       #MyWord := W#0;
       #MyBoolsinWord[8] := #"EMUOK";    //EPICSName: EMUOK
       #MyBoolsinWord[9] := #"EMUOK_Magtr";    //EPICSName: EMUOK_Magtr
       "PLCToEPICS"."Word"[#PLCToEPICSDataBlockOffset + 0] := #MyWord;
    Else
       #DEVICE_PARAM_OK := FALSE; //Invalid Hash
    END_IF;
END_FUNCTION_BLOCK
FUNCTION_BLOCK "DEVTYPE_ISRC_LEBT_INTF_HMI"
{ S7_Optimized_Access := 'TRUE' }
VERSION : 1.0
   VAR_INPUT
      "ComIocOK" { ExternalAccessible := 'True'; ExternalVisible := 'False'; ExternalWritable := 'False'; } : BOOL;   //EPICS Status variable: ComIocOK
      "ComRioOK" { ExternalAccessible := 'True'; ExternalVisible := 'False'; ExternalWritable := 'False'; } : BOOL;   //EPICS Status variable: ComRioOK
      "ISrcOK" { ExternalAccessible := 'True'; ExternalVisible := 'False'; ExternalWritable := 'False'; } : BOOL;   //EPICS Status variable: ISrcOK
      "EVENT_A_MEMO" { ExternalAccessible := 'True'; ExternalVisible := 'False'; ExternalWritable := 'False'; } : BOOL;   //EPICS Status variable: EVENT_A_MEMO
      "EVENT_B_MEMO" { ExternalAccessible := 'True'; ExternalVisible := 'False'; ExternalWritable := 'False'; } : BOOL;   //EPICS Status variable: EVENT_B_MEMO
      "EVENT_C_MEMO" { ExternalAccessible := 'True'; ExternalVisible := 'False'; ExternalWritable := 'False'; } : BOOL;   //EPICS Status variable: EVENT_C_MEMO
      "EVENT_D_MEMO" { ExternalAccessible := 'True'; ExternalVisible := 'False'; ExternalWritable := 'False'; } : BOOL;   //EPICS Status variable: EVENT_D_MEMO
      "EVENT_E_MEMO" { ExternalAccessible := 'True'; ExternalVisible := 'False'; ExternalWritable := 'False'; } : BOOL;   //EPICS Status variable: EVENT_E_MEMO
      "EVENT_F_MEMO" { ExternalAccessible := 'True'; ExternalVisible := 'False'; ExternalWritable := 'False'; } : BOOL;   //EPICS Status variable: EVENT_F_MEMO
      "EVENT_G_MEMO" { ExternalAccessible := 'True'; ExternalVisible := 'False'; ExternalWritable := 'False'; } : BOOL;   //EPICS Status variable: EVENT_G_MEMO
      "EVENT_H_MEMO" { ExternalAccessible := 'True'; ExternalVisible := 'False'; ExternalWritable := 'False'; } : BOOL;   //EPICS Status variable: EVENT_H_MEMO
      "ChopPwrSysOK_MEMO" { ExternalAccessible := 'True'; ExternalVisible := 'False'; ExternalWritable := 'False'; } : BOOL;   //EPICS Status variable: ChopPwrSysOK_MEMO
      "ChopVoltAlarm_MEMO" { ExternalAccessible := 'True'; ExternalVisible := 'False'; ExternalWritable := 'False'; } : BOOL;   //EPICS Status variable: ChopVoltAlarm_MEMO
      "ChopWtrFlowOK_MEMO" { ExternalAccessible := 'True'; ExternalVisible := 'False'; ExternalWritable := 'False'; } : BOOL;   //EPICS Status variable: ChopWtrFlowOK_MEMO
      "Sol1WtrTempOK_MEMO" { ExternalAccessible := 'True'; ExternalVisible := 'False'; ExternalWritable := 'False'; } : BOOL;   //EPICS Status variable: Sol1WtrTempOK_MEMO
      "Sol2WtrTempOK_MEMO" { ExternalAccessible := 'True'; ExternalVisible := 'False'; ExternalWritable := 'False'; } : BOOL;   //EPICS Status variable: Sol2WtrTempOK_MEMO
      "Sol1WtrFlowOK_MEMO" { ExternalAccessible := 'True'; ExternalVisible := 'False'; ExternalWritable := 'False'; } : BOOL;   //EPICS Status variable: Sol1WtrFlowOK_MEMO
      "Sol2WtrFlowOK_MEMO" { ExternalAccessible := 'True'; ExternalVisible := 'False'; ExternalWritable := 'False'; } : BOOL;   //EPICS Status variable: Sol2WtrFlowOK_MEMO
      "Sol1CurMaxErr_MEMO" { ExternalAccessible := 'True'; ExternalVisible := 'False'; ExternalWritable := 'False'; } : BOOL;   //EPICS Status variable: Sol1CurMaxErr_MEMO
      "Sol2CurMaxErr_MEMO" { ExternalAccessible := 'True'; ExternalVisible := 'False'; ExternalWritable := 'False'; } : BOOL;   //EPICS Status variable: Sol2CurMaxErr_MEMO
      "Str1HCurMaxErr_MEMO" { ExternalAccessible := 'True'; ExternalVisible := 'False'; ExternalWritable := 'False'; } : BOOL;   //EPICS Status variable: Str1HCurMaxErr_MEMO
      "Str2HCurMaxErr_MEMO" { ExternalAccessible := 'True'; ExternalVisible := 'False'; ExternalWritable := 'False'; } : BOOL;   //EPICS Status variable: Str2HCurMaxErr_MEMO
      "Str1VCurMaxErr_MEMO" { ExternalAccessible := 'True'; ExternalVisible := 'False'; ExternalWritable := 'False'; } : BOOL;   //EPICS Status variable: Str1VCurMaxErr_MEMO
      "Str2VCurMaxErr_MEMO" { ExternalAccessible := 'True'; ExternalVisible := 'False'; ExternalWritable := 'False'; } : BOOL;   //EPICS Status variable: Str2VCurMaxErr_MEMO
      "Coil1PwrSuppOK_MEMO" { ExternalAccessible := 'True'; ExternalVisible := 'False'; ExternalWritable := 'False'; } : BOOL;   //EPICS Status variable: Coil1PwrSuppOK_MEMO
      "Coil2PwrSuppOK_MEMO" { ExternalAccessible := 'True'; ExternalVisible := 'False'; ExternalWritable := 'False'; } : BOOL;   //EPICS Status variable: Coil2PwrSuppOK_MEMO
      "Coil3PwrSuppOK_MEMO" { ExternalAccessible := 'True'; ExternalVisible := 'False'; ExternalWritable := 'False'; } : BOOL;   //EPICS Status variable: Coil3PwrSuppOK_MEMO
      "HVITLidOpenR_MEMO" { ExternalAccessible := 'True'; ExternalVisible := 'False'; ExternalWritable := 'False'; } : BOOL;   //EPICS Status variable: HVITLidOpenR_MEMO
      "HVITOilTempOK_MEMO" { ExternalAccessible := 'True'; ExternalVisible := 'False'; ExternalWritable := 'False'; } : BOOL;   //EPICS Status variable: HVITOilTempOK_MEMO
      "GndWtrTempMaxErr_MEMO" { ExternalAccessible := 'True'; ExternalVisible := 'False'; ExternalWritable := 'False'; } : BOOL;   //EPICS Status variable: GndWtrTempMaxErr_MEMO
      "HVWtrTempMaxErr_MEMO" { ExternalAccessible := 'True'; ExternalVisible := 'False'; ExternalWritable := 'False'; } : BOOL;   //EPICS Status variable: HVWtrTempMaxErr_MEMO
      "RepWtrFlowOK_MEMO" { ExternalAccessible := 'True'; ExternalVisible := 'False'; ExternalWritable := 'False'; } : BOOL;   //EPICS Status variable: RepWtrFlowOK_MEMO
      "IrisWtrTemp1Err_MEMO" { ExternalAccessible := 'True'; ExternalVisible := 'False'; ExternalWritable := 'False'; } : BOOL;   //EPICS Status variable: IrisWtrTemp1Err_MEMO
      "IrisWtrTemp2Err_MEMO" { ExternalAccessible := 'True'; ExternalVisible := 'False'; ExternalWritable := 'False'; } : BOOL;   //EPICS Status variable: IrisWtrTemp2Err_MEMO
      "IrisWtrFlowOK_MEMO" { ExternalAccessible := 'True'; ExternalVisible := 'False'; ExternalWritable := 'False'; } : BOOL;   //EPICS Status variable: IrisWtrFlowOK_MEMO
      "EMUHWtrFlowOK_MEMO" { ExternalAccessible := 'True'; ExternalVisible := 'False'; ExternalWritable := 'False'; } : BOOL;   //EPICS Status variable: EMUHWtrFlowOK_MEMO
      "EMUVWtrFlowOK_MEMO" { ExternalAccessible := 'True'; ExternalVisible := 'False'; ExternalWritable := 'False'; } : BOOL;   //EPICS Status variable: EMUVWtrFlowOK_MEMO
      "FCWtrFlowOK_MEMO" { ExternalAccessible := 'True'; ExternalVisible := 'False'; ExternalWritable := 'False'; } : BOOL;   //EPICS Status variable: FCWtrFlowOK_MEMO
      "EMUOK_MEMO" { ExternalAccessible := 'True'; ExternalVisible := 'False'; ExternalWritable := 'False'; } : BOOL;   //EPICS Status variable: EMUOK_MEMO
      "IBSWtrFlowOK_MEMO" { ExternalAccessible := 'True'; ExternalVisible := 'False'; ExternalWritable := 'False'; } : BOOL;   //EPICS Status variable: IBSWtrFlowOK_MEMO
      "CollWtrFlowOK_MEMO" { ExternalAccessible := 'True'; ExternalVisible := 'False'; ExternalWritable := 'False'; } : BOOL;   //EPICS Status variable: CollWtrFlowOK_MEMO
      "MatTrWtrFlowOK_MEMO" { ExternalAccessible := 'True'; ExternalVisible := 'False'; ExternalWritable := 'False'; } : BOOL;   //EPICS Status variable: MatTrWtrFlowOK_MEMO
      "PlasChWtrFlowOK_MEMO" { ExternalAccessible := 'True'; ExternalVisible := 'False'; ExternalWritable := 'False'; } : BOOL;   //EPICS Status variable: PlasChWtrFlowOK_MEMO
      "VacOK_MEMO" { ExternalAccessible := 'True'; ExternalVisible := 'False'; ExternalWritable := 'False'; } : BOOL;   //EPICS Status variable: VacOK_MEMO
      "VacPermit_MEMO" { ExternalAccessible := 'True'; ExternalVisible := 'False'; ExternalWritable := 'False'; } : BOOL;   //EPICS Status variable: VacPermit_MEMO
      "ComRioOK_MEMO" { ExternalAccessible := 'True'; ExternalVisible := 'False'; ExternalWritable := 'False'; } : BOOL;   //EPICS Status variable: ComRioOK_MEMO
      "MPSOK_MEMO" { ExternalAccessible := 'True'; ExternalVisible := 'False'; ExternalWritable := 'False'; } : BOOL;   //EPICS Status variable: MPSOK_MEMO
      "HVPSVolOK_Magtr_MEMO" { ExternalAccessible := 'True'; ExternalVisible := 'False'; ExternalWritable := 'False'; } : BOOL;   //EPICS Status variable: HVPSVolOK_Magtr_MEMO
      "DPLOK_MEMO" { ExternalAccessible := 'True'; ExternalVisible := 'False'; ExternalWritable := 'False'; } : BOOL;   //EPICS Status variable: DPLOK_MEMO
      "HVPfDoors_MEMO" { ExternalAccessible := 'True'; ExternalVisible := 'False'; ExternalWritable := 'False'; } : BOOL;   //EPICS Status variable: HVPfDoors_MEMO
      "HVPfRes_MEMO" { ExternalAccessible := 'True'; ExternalVisible := 'False'; ExternalWritable := 'False'; } : BOOL;   //EPICS Status variable: HVPfRes_MEMO
      "HVPermit_MEMO" { ExternalAccessible := 'True'; ExternalVisible := 'False'; ExternalWritable := 'False'; } : BOOL;   //EPICS Status variable: HVPermit_MEMO
      "ComIocOK_MEMO" { ExternalAccessible := 'True'; ExternalVisible := 'False'; ExternalWritable := 'False'; } : BOOL;   //EPICS Status variable: ComIocOK_MEMO
      "Rep1VolOK_MEMO" { ExternalAccessible := 'True'; ExternalVisible := 'False'; ExternalWritable := 'False'; } : BOOL;   //EPICS Status variable: Rep1VolOK_MEMO
      "Rep2VolOK_MEMO" { ExternalAccessible := 'True'; ExternalVisible := 'False'; ExternalWritable := 'False'; } : BOOL;   //EPICS Status variable: Rep2VolOK_MEMO
      "MagPulseModeOK_MEMO" { ExternalAccessible := 'True'; ExternalVisible := 'False'; ExternalWritable := 'False'; } : BOOL;   //EPICS Status variable: MagPulseModeOK_MEMO
      "ESTOP_MEMO" { ExternalAccessible := 'True'; ExternalVisible := 'False'; ExternalWritable := 'False'; } : BOOL;   //EPICS Status variable: ESTOP_MEMO
      "HVPSConnErr_MEMO" { ExternalAccessible := 'True'; ExternalVisible := 'False'; ExternalWritable := 'False'; } : BOOL;   //EPICS Status variable: HVPSConnErr_MEMO
      "Coil1WtrFlowOK_MEMO" { ExternalAccessible := 'True'; ExternalVisible := 'False'; ExternalWritable := 'False'; } : BOOL;   //EPICS Status variable: Coil1WtrFlowOK_MEMO
      "Coil2WtrFlowOK_MEMO" { ExternalAccessible := 'True'; ExternalVisible := 'False'; ExternalWritable := 'False'; } : BOOL;   //EPICS Status variable: Coil2WtrFlowOK_MEMO
      "Coil3WtrFlowOK_MEMO" { ExternalAccessible := 'True'; ExternalVisible := 'False'; ExternalWritable := 'False'; } : BOOL;   //EPICS Status variable: Coil3WtrFlowOK_MEMO
      "Coil1WtrTempOK_MEMO" { ExternalAccessible := 'True'; ExternalVisible := 'False'; ExternalWritable := 'False'; } : BOOL;   //EPICS Status variable: Coil1WtrTempOK_MEMO
      "Coil2WtrTempOK_MEMO" { ExternalAccessible := 'True'; ExternalVisible := 'False'; ExternalWritable := 'False'; } : BOOL;   //EPICS Status variable: Coil2WtrTempOK_MEMO
      "Coil3WtrTempOK_MEMO" { ExternalAccessible := 'True'; ExternalVisible := 'False'; ExternalWritable := 'False'; } : BOOL;   //EPICS Status variable: Coil3WtrTempOK_MEMO
      "F_MagtrEnCmd" { ExternalAccessible := 'True'; ExternalVisible := 'False'; ExternalWritable := 'False'; } : BOOL;   //EPICS Status variable: F_MagtrEnCmd
      "F_ChopWtrFlowOK" { ExternalAccessible := 'True'; ExternalVisible := 'False'; ExternalWritable := 'False'; } : BOOL;   //EPICS Status variable: F_ChopWtrFlowOK
      "F_ChopPwrSysOK" { ExternalAccessible := 'True'; ExternalVisible := 'False'; ExternalWritable := 'False'; } : BOOL;   //EPICS Status variable: F_ChopPwrSysOK
      "F_ChopVoltAlarm" { ExternalAccessible := 'True'; ExternalVisible := 'False'; ExternalWritable := 'False'; } : BOOL;   //EPICS Status variable: F_ChopVoltAlarm
      "F_Sol1WtrTempOK" { ExternalAccessible := 'True'; ExternalVisible := 'False'; ExternalWritable := 'False'; } : BOOL;   //EPICS Status variable: F_Sol1WtrTempOK
      "F_Sol2WtrTempOK" { ExternalAccessible := 'True'; ExternalVisible := 'False'; ExternalWritable := 'False'; } : BOOL;   //EPICS Status variable: F_Sol2WtrTempOK
      "F_Sol1WtrFlowOK" { ExternalAccessible := 'True'; ExternalVisible := 'False'; ExternalWritable := 'False'; } : BOOL;   //EPICS Status variable: F_Sol1WtrFlowOK
      "F_Sol2WtrFlowOK" { ExternalAccessible := 'True'; ExternalVisible := 'False'; ExternalWritable := 'False'; } : BOOL;   //EPICS Status variable: F_Sol2WtrFlowOK
      "F_Sol1CurMaxErr" { ExternalAccessible := 'True'; ExternalVisible := 'False'; ExternalWritable := 'False'; } : BOOL;   //EPICS Status variable: F_Sol1CurMaxErr
      "F_Sol2CurMaxErr" { ExternalAccessible := 'True'; ExternalVisible := 'False'; ExternalWritable := 'False'; } : BOOL;   //EPICS Status variable: F_Sol2CurMaxErr
      "F_Str1HCurMaxErr" { ExternalAccessible := 'True'; ExternalVisible := 'False'; ExternalWritable := 'False'; } : BOOL;   //EPICS Status variable: F_Str1HCurMaxErr
      "F_Str2HCurMaxErr" { ExternalAccessible := 'True'; ExternalVisible := 'False'; ExternalWritable := 'False'; } : BOOL;   //EPICS Status variable: F_Str2HCurMaxErr
      "F_Str1VCurMaxErr" { ExternalAccessible := 'True'; ExternalVisible := 'False'; ExternalWritable := 'False'; } : BOOL;   //EPICS Status variable: F_Str1VCurMaxErr
      "F_Str2VCurMaxErr" { ExternalAccessible := 'True'; ExternalVisible := 'False'; ExternalWritable := 'False'; } : BOOL;   //EPICS Status variable: F_Str2VCurMaxErr
      "F_Coil1WtrFlowOK" { ExternalAccessible := 'True'; ExternalVisible := 'False'; ExternalWritable := 'False'; } : BOOL;   //EPICS Status variable: F_Coil1WtrFlowOK
      "F_Coil2WtrFlowOK" { ExternalAccessible := 'True'; ExternalVisible := 'False'; ExternalWritable := 'False'; } : BOOL;   //EPICS Status variable: F_Coil2WtrFlowOK
      "F_Coil3WtrFlowOK" { ExternalAccessible := 'True'; ExternalVisible := 'False'; ExternalWritable := 'False'; } : BOOL;   //EPICS Status variable: F_Coil3WtrFlowOK
      "F_Coil1WtrTempOK" { ExternalAccessible := 'True'; ExternalVisible := 'False'; ExternalWritable := 'False'; } : BOOL;   //EPICS Status variable: F_Coil1WtrTempOK
      "F_Coil2WtrTempOK" { ExternalAccessible := 'True'; ExternalVisible := 'False'; ExternalWritable := 'False'; } : BOOL;   //EPICS Status variable: F_Coil2WtrTempOK
      "F_Coil3WtrTempOK" { ExternalAccessible := 'True'; ExternalVisible := 'False'; ExternalWritable := 'False'; } : BOOL;   //EPICS Status variable: F_Coil3WtrTempOK
      "F_Coil1PwrSuppOK" { ExternalAccessible := 'True'; ExternalVisible := 'False'; ExternalWritable := 'False'; } : BOOL;   //EPICS Status variable: F_Coil1PwrSuppOK
      "F_Coil2PwrSuppOK" { ExternalAccessible := 'True'; ExternalVisible := 'False'; ExternalWritable := 'False'; } : BOOL;   //EPICS Status variable: F_Coil2PwrSuppOK
      "F_Coil3PwrSuppOK" { ExternalAccessible := 'True'; ExternalVisible := 'False'; ExternalWritable := 'False'; } : BOOL;   //EPICS Status variable: F_Coil3PwrSuppOK
      "F_HVITLidOpen" { ExternalAccessible := 'True'; ExternalVisible := 'False'; ExternalWritable := 'False'; } : BOOL;   //EPICS Status variable: F_HVITLidOpen
      "F_HVITOilTempOK" { ExternalAccessible := 'True'; ExternalVisible := 'False'; ExternalWritable := 'False'; } : BOOL;   //EPICS Status variable: F_HVITOilTempOK
      "F_GndWtrTempMaxErr" { ExternalAccessible := 'True'; ExternalVisible := 'False'; ExternalWritable := 'False'; } : BOOL;   //EPICS Status variable: F_GndWtrTempMaxErr
      "F_HVWtrTempMaxErr" { ExternalAccessible := 'True'; ExternalVisible := 'False'; ExternalWritable := 'False'; } : BOOL;   //EPICS Status variable: F_HVWtrTempMaxErr
      "F_RepWtrFlowOK" { ExternalAccessible := 'True'; ExternalVisible := 'False'; ExternalWritable := 'False'; } : BOOL;   //EPICS Status variable: F_RepWtrFlowOK
      "F_Rep1VolOK" { ExternalAccessible := 'True'; ExternalVisible := 'False'; ExternalWritable := 'False'; } : BOOL;   //EPICS Status variable: F_Rep1VolOK
      "F_Rep2VolOK" { ExternalAccessible := 'True'; ExternalVisible := 'False'; ExternalWritable := 'False'; } : BOOL;   //EPICS Status variable: F_Rep2VolOK
      "F_IrisWtrTemp1Err" { ExternalAccessible := 'True'; ExternalVisible := 'False'; ExternalWritable := 'False'; } : BOOL;   //EPICS Status variable: F_IrisWtrTemp1Err
      "F_IrisWtrTemp2Err" { ExternalAccessible := 'True'; ExternalVisible := 'False'; ExternalWritable := 'False'; } : BOOL;   //EPICS Status variable: F_IrisWtrTemp2Err
      "F_IrisWtrFlowOK" { ExternalAccessible := 'True'; ExternalVisible := 'False'; ExternalWritable := 'False'; } : BOOL;   //EPICS Status variable: F_IrisWtrFlowOK
      "F_FCWtrFlowOK" { ExternalAccessible := 'True'; ExternalVisible := 'False'; ExternalWritable := 'False'; } : BOOL;   //EPICS Status variable: F_FCWtrFlowOK
      "F_EMUHWtrFlowOK" { ExternalAccessible := 'True'; ExternalVisible := 'False'; ExternalWritable := 'False'; } : BOOL;   //EPICS Status variable: F_EMUHWtrFlowOK
      "F_EMUVWtrFlowOK" { ExternalAccessible := 'True'; ExternalVisible := 'False'; ExternalWritable := 'False'; } : BOOL;   //EPICS Status variable: F_EMUVWtrFlowOK
      "F_EMUOK" { ExternalAccessible := 'True'; ExternalVisible := 'False'; ExternalWritable := 'False'; } : BOOL;   //EPICS Status variable: F_EMUOK
      "F_IBSWtrFlowOK" { ExternalAccessible := 'True'; ExternalVisible := 'False'; ExternalWritable := 'False'; } : BOOL;   //EPICS Status variable: F_IBSWtrFlowOK
      "F_CollWtrFlowOK" { ExternalAccessible := 'True'; ExternalVisible := 'False'; ExternalWritable := 'False'; } : BOOL;   //EPICS Status variable: F_CollWtrFlowOK
      "F_MatTrWtrFlowOK" { ExternalAccessible := 'True'; ExternalVisible := 'False'; ExternalWritable := 'False'; } : BOOL;   //EPICS Status variable: F_MatTrWtrFlowOK
      "F_PlasChWtrFlowOK" { ExternalAccessible := 'True'; ExternalVisible := 'False'; ExternalWritable := 'False'; } : BOOL;   //EPICS Status variable: F_PlasChWtrFlowOK
      "F_ComRioOK" { ExternalAccessible := 'True'; ExternalVisible := 'False'; ExternalWritable := 'False'; } : BOOL;   //EPICS Status variable: F_ComRioOK
      "F_MPSOK" { ExternalAccessible := 'True'; ExternalVisible := 'False'; ExternalWritable := 'False'; } : BOOL;   //EPICS Status variable: F_MPSOK
      "F_VacOK" { ExternalAccessible := 'True'; ExternalVisible := 'False'; ExternalWritable := 'False'; } : BOOL;   //EPICS Status variable: F_VacOK
      "F_VacPermit" { ExternalAccessible := 'True'; ExternalVisible := 'False'; ExternalWritable := 'False'; } : BOOL;   //EPICS Status variable: F_VacPermit
      "F_HVPSVolOK_Magtr" { ExternalAccessible := 'True'; ExternalVisible := 'False'; ExternalWritable := 'False'; } : BOOL;   //EPICS Status variable: F_HVPSVolOK_Magtr
      "F_MagPulseModeOK" { ExternalAccessible := 'True'; ExternalVisible := 'False'; ExternalWritable := 'False'; } : BOOL;   //EPICS Status variable: F_MagPulseModeOK
      "F_DPLOK" { ExternalAccessible := 'True'; ExternalVisible := 'False'; ExternalWritable := 'False'; } : BOOL;   //EPICS Status variable: F_DPLOK
      "F_HVITLckEnCmd" { ExternalAccessible := 'True'; ExternalVisible := 'False'; ExternalWritable := 'False'; } : BOOL;   //EPICS Status variable: F_HVITLckEnCmd
      "F_HVPfDoors" { ExternalAccessible := 'True'; ExternalVisible := 'False'; ExternalWritable := 'False'; } : BOOL;   //EPICS Status variable: F_HVPfDoors
      "F_HVPfRes" { ExternalAccessible := 'True'; ExternalVisible := 'False'; ExternalWritable := 'False'; } : BOOL;   //EPICS Status variable: F_HVPfRes
      "F_HVPermit" { ExternalAccessible := 'True'; ExternalVisible := 'False'; ExternalWritable := 'False'; } : BOOL;   //EPICS Status variable: F_HVPermit
      "F_ComIocOK" { ExternalAccessible := 'True'; ExternalVisible := 'False'; ExternalWritable := 'False'; } : BOOL;   //EPICS Status variable: F_ComIocOK
      "F_Coil1EnCmd" { ExternalAccessible := 'True'; ExternalVisible := 'False'; ExternalWritable := 'False'; } : BOOL;   //EPICS Status variable: F_Coil1EnCmd
      "F_Coil2EnCmd" { ExternalAccessible := 'True'; ExternalVisible := 'False'; ExternalWritable := 'False'; } : BOOL;   //EPICS Status variable: F_Coil2EnCmd
      "F_Coil3EnCmd" { ExternalAccessible := 'True'; ExternalVisible := 'False'; ExternalWritable := 'False'; } : BOOL;   //EPICS Status variable: F_Coil3EnCmd
      "F_Sol1EnCmd" { ExternalAccessible := 'True'; ExternalVisible := 'False'; ExternalWritable := 'False'; } : BOOL;   //EPICS Status variable: F_Sol1EnCmd
      "F_Str1HEnCmd" { ExternalAccessible := 'True'; ExternalVisible := 'False'; ExternalWritable := 'False'; } : BOOL;   //EPICS Status variable: F_Str1HEnCmd
      "F_Str1VEnCmd" { ExternalAccessible := 'True'; ExternalVisible := 'False'; ExternalWritable := 'False'; } : BOOL;   //EPICS Status variable: F_Str1VEnCmd
      "F_Sol2EnCmd" { ExternalAccessible := 'True'; ExternalVisible := 'False'; ExternalWritable := 'False'; } : BOOL;   //EPICS Status variable: F_Sol2EnCmd
      "F_Str2HEnCmd" { ExternalAccessible := 'True'; ExternalVisible := 'False'; ExternalWritable := 'False'; } : BOOL;   //EPICS Status variable: F_Str2HEnCmd
      "F_Str2VEnCmd" { ExternalAccessible := 'True'; ExternalVisible := 'False'; ExternalWritable := 'False'; } : BOOL;   //EPICS Status variable: F_Str2VEnCmd
      "F_VacVVAOpenCmd" { ExternalAccessible := 'True'; ExternalVisible := 'False'; ExternalWritable := 'False'; } : BOOL;   //EPICS Status variable: F_VacVVAOpenCmd
      "F_ChopHVEnCmd" { ExternalAccessible := 'True'; ExternalVisible := 'False'; ExternalWritable := 'False'; } : BOOL;   //EPICS Status variable: F_ChopHVEnCmd
      "F_ISrcOKtoMPS" { ExternalAccessible := 'True'; ExternalVisible := 'False'; ExternalWritable := 'False'; } : BOOL;   //EPICS Status variable: F_ISrcOKtoMPS
      "F_MWPowerOn" { ExternalAccessible := 'True'; ExternalVisible := 'False'; ExternalWritable := 'False'; } : BOOL;   //EPICS Status variable: F_MWPowerOn
      "F_VacVEVMCOK" { ExternalAccessible := 'True'; ExternalVisible := 'False'; ExternalWritable := 'False'; } : BOOL;   //EPICS Status variable: F_VacVEVMCOK
      "F_GNDInletPres" { ExternalAccessible := 'True'; ExternalVisible := 'False'; ExternalWritable := 'False'; } : BOOL;   //EPICS Status variable: F_GNDInletPres
      "F_GNDOutletPres" { ExternalAccessible := 'True'; ExternalVisible := 'False'; ExternalWritable := 'False'; } : BOOL;   //EPICS Status variable: F_GNDOutletPres
   EPICSToPLCLength { ExternalAccessible := 'False'; ExternalVisible := 'False'; ExternalWritable := 'False'; } : Int;   // Length of device command register array (in words)
   EPICSToPLCDataBlockOffset { ExternalAccessible := 'False'; ExternalVisible := 'False'; ExternalWritable := 'False'; } : Int;   // Offset in EPICS->PLC comms block where this device data resides (in words)
   EPICSToPLCParametersStart { ExternalAccessible := 'False'; ExternalVisible := 'False'; ExternalWritable := 'False'; } : Int;   // The border offset between the Command and the Parameter area
   PLCToEPICSLength { ExternalAccessible := 'False'; ExternalVisible := 'False'; ExternalWritable := 'False'; } : Int;   // Length of device status register array (in words)
   PLCToEPICSDataBlockOffset { ExternalAccessible := 'False'; ExternalVisible := 'False'; ExternalWritable := 'False'; } : Int;   // Offset in PLC->EPICS comms block where this device data resides (in words)
   END_VAR
   VAR_OUTPUT
      "EVENT_A_ACK" { ExternalAccessible := 'True'; ExternalVisible := 'False'; ExternalWritable := 'False'; } : BOOL;   //EPICS Command variable: EVENT_A_ACK
      "EVENT_B_ACK" { ExternalAccessible := 'True'; ExternalVisible := 'False'; ExternalWritable := 'False'; } : BOOL;   //EPICS Command variable: EVENT_B_ACK
      "EVENT_C_ACK" { ExternalAccessible := 'True'; ExternalVisible := 'False'; ExternalWritable := 'False'; } : BOOL;   //EPICS Command variable: EVENT_C_ACK
      "EVENT_D_ACK" { ExternalAccessible := 'True'; ExternalVisible := 'False'; ExternalWritable := 'False'; } : BOOL;   //EPICS Command variable: EVENT_D_ACK
      "EVENT_E_ACK" { ExternalAccessible := 'True'; ExternalVisible := 'False'; ExternalWritable := 'False'; } : BOOL;   //EPICS Command variable: EVENT_E_ACK
      "EVENT_F_ACK" { ExternalAccessible := 'True'; ExternalVisible := 'False'; ExternalWritable := 'False'; } : BOOL;   //EPICS Command variable: EVENT_F_ACK
      "EVENT_G_ACK" { ExternalAccessible := 'True'; ExternalVisible := 'False'; ExternalWritable := 'False'; } : BOOL;   //EPICS Command variable: EVENT_G_ACK
      "EVENT_H_ACK" { ExternalAccessible := 'True'; ExternalVisible := 'False'; ExternalWritable := 'False'; } : BOOL;   //EPICS Command variable: EVENT_H_ACK
      "VacLevelMaxS" { ExternalAccessible := 'True'; ExternalVisible := 'False'; ExternalWritable := 'False'; } : REAL;   //EPICS Parameter variable: VacLevelMaxS
      DEVICE_PARAM_OK { ExternalAccessible := 'False'; ExternalVisible := 'False'; ExternalWritable := 'False'; } : Bool;
   END_VAR
   VAR_IN_OUT
   END_VAR
   Var DB_SPECIFIC
      MyWord { ExternalAccessible := 'False'; ExternalVisible := 'False'; ExternalWritable := 'False'; } : Word;
      MyBytesinWord { ExternalAccessible := 'False'; ExternalVisible := 'False'; ExternalWritable := 'False'; } AT MyWord : Array[0..1] of Byte;
      MyBoolsinWord { ExternalAccessible := 'False'; ExternalVisible := 'False'; ExternalWritable := 'False'; } AT MyWord : Array[0..15] of Bool;
      MyDInt { ExternalAccessible := 'False'; ExternalVisible := 'False'; ExternalWritable := 'False'; } : DInt;
      MyWordsinDint { ExternalAccessible := 'False'; ExternalVisible := 'False'; ExternalWritable := 'False'; } AT MyDInt : Array[0..1] of Word;
      MyReal { ExternalAccessible := 'False'; ExternalVisible := 'False'; ExternalWritable := 'False'; } : Real;
      MyWordsinReal { ExternalAccessible := 'False'; ExternalVisible := 'False'; ExternalWritable := 'False'; } AT MyReal : Array[0..1] of Word;
      MyInt { ExternalAccessible := 'False'; ExternalVisible := 'False'; ExternalWritable := 'False'; } : Int;
      MyWordinInt { ExternalAccessible := 'False'; ExternalVisible := 'False'; ExternalWritable := 'False'; } AT MyInt : Word;
      MyDWord { ExternalAccessible := 'False'; ExternalVisible := 'False'; ExternalWritable := 'False'; } : DWord;
      MyWordsinDWord { ExternalAccessible := 'False'; ExternalVisible := 'False'; ExternalWritable := 'False'; } AT MyDWord : Array[0..1] of Word;
      MyTime { ExternalAccessible := 'False'; ExternalVisible := 'False'; ExternalWritable := 'False'; } : Time;
      MyWordsinTime { ExternalAccessible := 'False'; ExternalVisible := 'False'; ExternalWritable := 'False'; } AT MyTime : Array[0..1] of Word;
      MyString { ExternalAccessible := 'False'; ExternalVisible := 'False'; ExternalWritable := 'False'; } : String[40];
      MyWordsinString { ExternalAccessible := 'False'; ExternalVisible := 'False'; ExternalWritable := 'False'; } AT MyString : Array[0..20] of Word;
   END_VAR
   VAR_TEMP
      HashModbus : DInt;
      HashIFA : DInt;
      HashTIAMap : DInt;
      i : Int;
   END_VAR
    //Author: Miklos Boros (miklos.boros@esss.se), Copyrigth 2017-2019 by European Spallation Source, Lund
    //This block was generated by PLCFactory, please don't change it MANUALLY!
    //Input File Name: ISrc-010_Ctrl-PLC-01-template-IFA-20191106135317.ifa
    //Generated: 20191106135317
    //According to HASH: 1347332123
    //Device type: ISRC_LEBT_INTF_HMI
    //Description: This function does the variable mapping for a device. All device-variable will be linked to an interface variable defined in this block.

    //********************************************
    //****************HASH check******************
    //********************************************


    #MyWordsinDint[0] := "EPICSToPLC"."Word"[0];
    #MyWordsinDint[1] := "EPICSToPLC"."Word"[1];
    #HashModbus := #MyDInt; //Hash from EPICS/ModbusTCP

    #HashIFA := 1347332123; //Hash from Interface Factory as a constant

    #MyWordsinDint[0] := "PLCToEPICS"."Word"[0];
    #MyWordsinDint[1] := "PLCToEPICS"."Word"[1];
    #HashTIAMap := #MyDInt; //Hash from PLCFactory TIA Map


    IF ((#HashIFA = #HashModbus) AND (#HashModbus = #HashTIAMap)) THEN //Check CRCs
        #DEVICE_PARAM_OK := TRUE;
       //###########################  ISRC_LEBT HMI  ##############################
       //###########################
       //STATUS BLOCK
       //###########################

    //********************************************
    //*************STATUS VARIABLES***************
    //********************************************


       #MyWord := W#0;
       #MyBoolsinWord[8] := #"ComIocOK";    //EPICSName: ComIocOK
       #MyBoolsinWord[9] := #"ComRioOK";    //EPICSName: ComRioOK
       #MyBoolsinWord[10] := #"ISrcOK";    //EPICSName: ISrcOK
       #MyBoolsinWord[11] := #"EVENT_A_MEMO";    //EPICSName: EVENT_A_MEMO
       #MyBoolsinWord[12] := #"EVENT_B_MEMO";    //EPICSName: EVENT_B_MEMO
       #MyBoolsinWord[13] := #"EVENT_C_MEMO";    //EPICSName: EVENT_C_MEMO
       #MyBoolsinWord[14] := #"EVENT_D_MEMO";    //EPICSName: EVENT_D_MEMO
       #MyBoolsinWord[15] := #"EVENT_E_MEMO";    //EPICSName: EVENT_E_MEMO
       #MyBoolsinWord[0] := #"EVENT_F_MEMO";    //EPICSName: EVENT_F_MEMO
       #MyBoolsinWord[1] := #"EVENT_G_MEMO";    //EPICSName: EVENT_G_MEMO
       #MyBoolsinWord[2] := #"EVENT_H_MEMO";    //EPICSName: EVENT_H_MEMO
       #MyBoolsinWord[3] := #"ChopPwrSysOK_MEMO";    //EPICSName: ChopPwrSysOK_MEMO
       #MyBoolsinWord[4] := #"ChopVoltAlarm_MEMO";    //EPICSName: ChopVoltAlarm_MEMO
       #MyBoolsinWord[5] := #"ChopWtrFlowOK_MEMO";    //EPICSName: ChopWtrFlowOK_MEMO
       #MyBoolsinWord[6] := #"Sol1WtrTempOK_MEMO";    //EPICSName: Sol1WtrTempOK_MEMO
       #MyBoolsinWord[7] := #"Sol2WtrTempOK_MEMO";    //EPICSName: Sol2WtrTempOK_MEMO
       "PLCToEPICS"."Word"[#PLCToEPICSDataBlockOffset + 0] := #MyWord;

       #MyWord := W#0;
       #MyBoolsinWord[8] := #"Sol1WtrFlowOK_MEMO";    //EPICSName: Sol1WtrFlowOK_MEMO
       #MyBoolsinWord[9] := #"Sol2WtrFlowOK_MEMO";    //EPICSName: Sol2WtrFlowOK_MEMO
       #MyBoolsinWord[10] := #"Sol1CurMaxErr_MEMO";    //EPICSName: Sol1CurMaxErr_MEMO
       #MyBoolsinWord[11] := #"Sol2CurMaxErr_MEMO";    //EPICSName: Sol2CurMaxErr_MEMO
       #MyBoolsinWord[12] := #"Str1HCurMaxErr_MEMO";    //EPICSName: Str1HCurMaxErr_MEMO
       #MyBoolsinWord[13] := #"Str2HCurMaxErr_MEMO";    //EPICSName: Str2HCurMaxErr_MEMO
       #MyBoolsinWord[14] := #"Str1VCurMaxErr_MEMO";    //EPICSName: Str1VCurMaxErr_MEMO
       #MyBoolsinWord[15] := #"Str2VCurMaxErr_MEMO";    //EPICSName: Str2VCurMaxErr_MEMO
       #MyBoolsinWord[0] := #"Coil1PwrSuppOK_MEMO";    //EPICSName: Coil1PwrSuppOK_MEMO
       #MyBoolsinWord[1] := #"Coil2PwrSuppOK_MEMO";    //EPICSName: Coil2PwrSuppOK_MEMO
       #MyBoolsinWord[2] := #"Coil3PwrSuppOK_MEMO";    //EPICSName: Coil3PwrSuppOK_MEMO
       #MyBoolsinWord[3] := #"HVITLidOpenR_MEMO";    //EPICSName: HVITLidOpenR_MEMO
       #MyBoolsinWord[4] := #"HVITOilTempOK_MEMO";    //EPICSName: HVITOilTempOK_MEMO
       #MyBoolsinWord[5] := #"GndWtrTempMaxErr_MEMO";    //EPICSName: GndWtrTempMaxErr_MEMO
       #MyBoolsinWord[6] := #"HVWtrTempMaxErr_MEMO";    //EPICSName: HVWtrTempMaxErr_MEMO
       #MyBoolsinWord[7] := #"RepWtrFlowOK_MEMO";    //EPICSName: RepWtrFlowOK_MEMO
       "PLCToEPICS"."Word"[#PLCToEPICSDataBlockOffset + 1] := #MyWord;

       #MyWord := W#0;
       #MyBoolsinWord[8] := #"IrisWtrTemp1Err_MEMO";    //EPICSName: IrisWtrTemp1Err_MEMO
       #MyBoolsinWord[9] := #"IrisWtrTemp2Err_MEMO";    //EPICSName: IrisWtrTemp2Err_MEMO
       #MyBoolsinWord[10] := #"IrisWtrFlowOK_MEMO";    //EPICSName: IrisWtrFlowOK_MEMO
       #MyBoolsinWord[11] := #"EMUHWtrFlowOK_MEMO";    //EPICSName: EMUHWtrFlowOK_MEMO
       #MyBoolsinWord[12] := #"EMUVWtrFlowOK_MEMO";    //EPICSName: EMUVWtrFlowOK_MEMO
       #MyBoolsinWord[13] := #"FCWtrFlowOK_MEMO";    //EPICSName: FCWtrFlowOK_MEMO
       #MyBoolsinWord[14] := #"EMUOK_MEMO";    //EPICSName: EMUOK_MEMO
       #MyBoolsinWord[15] := #"IBSWtrFlowOK_MEMO";    //EPICSName: IBSWtrFlowOK_MEMO
       #MyBoolsinWord[0] := #"CollWtrFlowOK_MEMO";    //EPICSName: CollWtrFlowOK_MEMO
       #MyBoolsinWord[1] := #"MatTrWtrFlowOK_MEMO";    //EPICSName: MatTrWtrFlowOK_MEMO
       #MyBoolsinWord[2] := #"PlasChWtrFlowOK_MEMO";    //EPICSName: PlasChWtrFlowOK_MEMO
       #MyBoolsinWord[3] := #"VacOK_MEMO";    //EPICSName: VacOK_MEMO
       #MyBoolsinWord[4] := #"VacPermit_MEMO";    //EPICSName: VacPermit_MEMO
       #MyBoolsinWord[5] := #"ComRioOK_MEMO";    //EPICSName: ComRioOK_MEMO
       #MyBoolsinWord[6] := #"MPSOK_MEMO";    //EPICSName: MPSOK_MEMO
       #MyBoolsinWord[7] := #"HVPSVolOK_Magtr_MEMO";    //EPICSName: HVPSVolOK_Magtr_MEMO
       "PLCToEPICS"."Word"[#PLCToEPICSDataBlockOffset + 2] := #MyWord;

       #MyWord := W#0;
       #MyBoolsinWord[8] := #"DPLOK_MEMO";    //EPICSName: DPLOK_MEMO
       #MyBoolsinWord[9] := #"HVPfDoors_MEMO";    //EPICSName: HVPfDoors_MEMO
       #MyBoolsinWord[10] := #"HVPfRes_MEMO";    //EPICSName: HVPfRes_MEMO
       #MyBoolsinWord[11] := #"HVPermit_MEMO";    //EPICSName: HVPermit_MEMO
       #MyBoolsinWord[12] := #"ComIocOK_MEMO";    //EPICSName: ComIocOK_MEMO
       #MyBoolsinWord[13] := #"Rep1VolOK_MEMO";    //EPICSName: Rep1VolOK_MEMO
       #MyBoolsinWord[14] := #"Rep2VolOK_MEMO";    //EPICSName: Rep2VolOK_MEMO
       #MyBoolsinWord[15] := #"MagPulseModeOK_MEMO";    //EPICSName: MagPulseModeOK_MEMO
       #MyBoolsinWord[0] := #"ESTOP_MEMO";    //EPICSName: ESTOP_MEMO
       #MyBoolsinWord[1] := #"HVPSConnErr_MEMO";    //EPICSName: HVPSConnErr_MEMO
       #MyBoolsinWord[2] := #"Coil1WtrFlowOK_MEMO";    //EPICSName: Coil1WtrFlowOK_MEMO
       #MyBoolsinWord[3] := #"Coil2WtrFlowOK_MEMO";    //EPICSName: Coil2WtrFlowOK_MEMO
       #MyBoolsinWord[4] := #"Coil3WtrFlowOK_MEMO";    //EPICSName: Coil3WtrFlowOK_MEMO
       #MyBoolsinWord[5] := #"Coil1WtrTempOK_MEMO";    //EPICSName: Coil1WtrTempOK_MEMO
       #MyBoolsinWord[6] := #"Coil2WtrTempOK_MEMO";    //EPICSName: Coil2WtrTempOK_MEMO
       #MyBoolsinWord[7] := #"Coil3WtrTempOK_MEMO";    //EPICSName: Coil3WtrTempOK_MEMO
       "PLCToEPICS"."Word"[#PLCToEPICSDataBlockOffset + 3] := #MyWord;

       #MyWord := W#0;
       #MyBoolsinWord[8] := #"F_MagtrEnCmd";    //EPICSName: F_MagtrEnCmd
       #MyBoolsinWord[9] := #"F_ChopWtrFlowOK";    //EPICSName: F_ChopWtrFlowOK
       #MyBoolsinWord[10] := #"F_ChopPwrSysOK";    //EPICSName: F_ChopPwrSysOK
       #MyBoolsinWord[11] := #"F_ChopVoltAlarm";    //EPICSName: F_ChopVoltAlarm
       #MyBoolsinWord[12] := #"F_Sol1WtrTempOK";    //EPICSName: F_Sol1WtrTempOK
       #MyBoolsinWord[13] := #"F_Sol2WtrTempOK";    //EPICSName: F_Sol2WtrTempOK
       #MyBoolsinWord[14] := #"F_Sol1WtrFlowOK";    //EPICSName: F_Sol1WtrFlowOK
       #MyBoolsinWord[15] := #"F_Sol2WtrFlowOK";    //EPICSName: F_Sol2WtrFlowOK
       #MyBoolsinWord[0] := #"F_Sol1CurMaxErr";    //EPICSName: F_Sol1CurMaxErr
       #MyBoolsinWord[1] := #"F_Sol2CurMaxErr";    //EPICSName: F_Sol2CurMaxErr
       #MyBoolsinWord[2] := #"F_Str1HCurMaxErr";    //EPICSName: F_Str1HCurMaxErr
       #MyBoolsinWord[3] := #"F_Str2HCurMaxErr";    //EPICSName: F_Str2HCurMaxErr
       #MyBoolsinWord[4] := #"F_Str1VCurMaxErr";    //EPICSName: F_Str1VCurMaxErr
       #MyBoolsinWord[5] := #"F_Str2VCurMaxErr";    //EPICSName: F_Str2VCurMaxErr
       #MyBoolsinWord[6] := #"F_Coil1WtrFlowOK";    //EPICSName: F_Coil1WtrFlowOK
       #MyBoolsinWord[7] := #"F_Coil2WtrFlowOK";    //EPICSName: F_Coil2WtrFlowOK
       "PLCToEPICS"."Word"[#PLCToEPICSDataBlockOffset + 4] := #MyWord;

       #MyWord := W#0;
       #MyBoolsinWord[8] := #"F_Coil3WtrFlowOK";    //EPICSName: F_Coil3WtrFlowOK
       #MyBoolsinWord[9] := #"F_Coil1WtrTempOK";    //EPICSName: F_Coil1WtrTempOK
       #MyBoolsinWord[10] := #"F_Coil2WtrTempOK";    //EPICSName: F_Coil2WtrTempOK
       #MyBoolsinWord[11] := #"F_Coil3WtrTempOK";    //EPICSName: F_Coil3WtrTempOK
       #MyBoolsinWord[12] := #"F_Coil1PwrSuppOK";    //EPICSName: F_Coil1PwrSuppOK
       #MyBoolsinWord[13] := #"F_Coil2PwrSuppOK";    //EPICSName: F_Coil2PwrSuppOK
       #MyBoolsinWord[14] := #"F_Coil3PwrSuppOK";    //EPICSName: F_Coil3PwrSuppOK
       #MyBoolsinWord[15] := #"F_HVITLidOpen";    //EPICSName: F_HVITLidOpen
       #MyBoolsinWord[0] := #"F_HVITOilTempOK";    //EPICSName: F_HVITOilTempOK
       #MyBoolsinWord[1] := #"F_GndWtrTempMaxErr";    //EPICSName: F_GndWtrTempMaxErr
       #MyBoolsinWord[2] := #"F_HVWtrTempMaxErr";    //EPICSName: F_HVWtrTempMaxErr
       #MyBoolsinWord[3] := #"F_RepWtrFlowOK";    //EPICSName: F_RepWtrFlowOK
       #MyBoolsinWord[4] := #"F_Rep1VolOK";    //EPICSName: F_Rep1VolOK
       #MyBoolsinWord[5] := #"F_Rep2VolOK";    //EPICSName: F_Rep2VolOK
       #MyBoolsinWord[6] := #"F_IrisWtrTemp1Err";    //EPICSName: F_IrisWtrTemp1Err
       #MyBoolsinWord[7] := #"F_IrisWtrTemp2Err";    //EPICSName: F_IrisWtrTemp2Err
       "PLCToEPICS"."Word"[#PLCToEPICSDataBlockOffset + 5] := #MyWord;

       #MyWord := W#0;
       #MyBoolsinWord[8] := #"F_IrisWtrFlowOK";    //EPICSName: F_IrisWtrFlowOK
       #MyBoolsinWord[9] := #"F_FCWtrFlowOK";    //EPICSName: F_FCWtrFlowOK
       #MyBoolsinWord[10] := #"F_EMUHWtrFlowOK";    //EPICSName: F_EMUHWtrFlowOK
       #MyBoolsinWord[11] := #"F_EMUVWtrFlowOK";    //EPICSName: F_EMUVWtrFlowOK
       #MyBoolsinWord[12] := #"F_EMUOK";    //EPICSName: F_EMUOK
       #MyBoolsinWord[13] := #"F_IBSWtrFlowOK";    //EPICSName: F_IBSWtrFlowOK
       #MyBoolsinWord[14] := #"F_CollWtrFlowOK";    //EPICSName: F_CollWtrFlowOK
       #MyBoolsinWord[15] := #"F_MatTrWtrFlowOK";    //EPICSName: F_MatTrWtrFlowOK
       #MyBoolsinWord[0] := #"F_PlasChWtrFlowOK";    //EPICSName: F_PlasChWtrFlowOK
       #MyBoolsinWord[1] := #"F_ComRioOK";    //EPICSName: F_ComRioOK
       #MyBoolsinWord[2] := #"F_MPSOK";    //EPICSName: F_MPSOK
       #MyBoolsinWord[3] := #"F_VacOK";    //EPICSName: F_VacOK
       #MyBoolsinWord[4] := #"F_VacPermit";    //EPICSName: F_VacPermit
       #MyBoolsinWord[5] := #"F_HVPSVolOK_Magtr";    //EPICSName: F_HVPSVolOK_Magtr
       #MyBoolsinWord[6] := #"F_MagPulseModeOK";    //EPICSName: F_MagPulseModeOK
       #MyBoolsinWord[7] := #"F_DPLOK";    //EPICSName: F_DPLOK
       "PLCToEPICS"."Word"[#PLCToEPICSDataBlockOffset + 6] := #MyWord;

       #MyWord := W#0;
       #MyBoolsinWord[8] := #"F_HVITLckEnCmd";    //EPICSName: F_HVITLckEnCmd
       #MyBoolsinWord[9] := #"F_HVPfDoors";    //EPICSName: F_HVPfDoors
       #MyBoolsinWord[10] := #"F_HVPfRes";    //EPICSName: F_HVPfRes
       #MyBoolsinWord[11] := #"F_HVPermit";    //EPICSName: F_HVPermit
       #MyBoolsinWord[12] := #"F_ComIocOK";    //EPICSName: F_ComIocOK
       #MyBoolsinWord[13] := #"F_Coil1EnCmd";    //EPICSName: F_Coil1EnCmd
       #MyBoolsinWord[14] := #"F_Coil2EnCmd";    //EPICSName: F_Coil2EnCmd
       #MyBoolsinWord[15] := #"F_Coil3EnCmd";    //EPICSName: F_Coil3EnCmd
       #MyBoolsinWord[0] := #"F_Sol1EnCmd";    //EPICSName: F_Sol1EnCmd
       #MyBoolsinWord[1] := #"F_Str1HEnCmd";    //EPICSName: F_Str1HEnCmd
       #MyBoolsinWord[2] := #"F_Str1VEnCmd";    //EPICSName: F_Str1VEnCmd
       #MyBoolsinWord[3] := #"F_Sol2EnCmd";    //EPICSName: F_Sol2EnCmd
       #MyBoolsinWord[4] := #"F_Str2HEnCmd";    //EPICSName: F_Str2HEnCmd
       #MyBoolsinWord[5] := #"F_Str2VEnCmd";    //EPICSName: F_Str2VEnCmd
       #MyBoolsinWord[6] := #"F_VacVVAOpenCmd";    //EPICSName: F_VacVVAOpenCmd
       #MyBoolsinWord[7] := #"F_ChopHVEnCmd";    //EPICSName: F_ChopHVEnCmd
       "PLCToEPICS"."Word"[#PLCToEPICSDataBlockOffset + 7] := #MyWord;

       #MyWord := W#0;
       #MyBoolsinWord[8] := #"F_ISrcOKtoMPS";    //EPICSName: F_ISrcOKtoMPS
       #MyBoolsinWord[9] := #"F_MWPowerOn";    //EPICSName: F_MWPowerOn
       #MyBoolsinWord[10] := #"F_VacVEVMCOK";    //EPICSName: F_VacVEVMCOK
       #MyBoolsinWord[11] := #"F_GNDInletPres";    //EPICSName: F_GNDInletPres
       #MyBoolsinWord[12] := #"F_GNDOutletPres";    //EPICSName: F_GNDOutletPres
       "PLCToEPICS"."Word"[#PLCToEPICSDataBlockOffset + 8] := #MyWord;

    //********************************************
    //*************COMMAND VARIABLES**************
    //********************************************


       #MyWord := "EPICSToPLC"."Word"[#EPICSToPLCDataBlockOffset + 0];
       IF (NOT "Utilities".TestInProgress) THEN
       	"EPICSToPLC"."Word"[#EPICSToPLCDataBlockOffset + 0] := 0;
       END_IF;
       #"EVENT_A_ACK" := #MyBoolsinWord[8];    //EPICSName: EVENT_A_ACK
       #"EVENT_B_ACK" := #MyBoolsinWord[9];    //EPICSName: EVENT_B_ACK
       #"EVENT_C_ACK" := #MyBoolsinWord[10];    //EPICSName: EVENT_C_ACK
       #"EVENT_D_ACK" := #MyBoolsinWord[11];    //EPICSName: EVENT_D_ACK
       #"EVENT_E_ACK" := #MyBoolsinWord[12];    //EPICSName: EVENT_E_ACK
       #"EVENT_F_ACK" := #MyBoolsinWord[13];    //EPICSName: EVENT_F_ACK
       #"EVENT_G_ACK" := #MyBoolsinWord[14];    //EPICSName: EVENT_G_ACK
       #"EVENT_H_ACK" := #MyBoolsinWord[15];    //EPICSName: EVENT_H_ACK

    //********************************************
    //************PARAMETER VARIABLES*************
    //********************************************


       #MyReal	:= 0.0;
       #MyWordsinReal[0]	:= "EPICSToPLC"."Word"[#EPICSToPLCDataBlockOffset + 1];
       #MyWordsinReal[1]	:= "EPICSToPLC"."Word"[#EPICSToPLCDataBlockOffset + 2];
       #"VacLevelMaxS" := #MyReal;    //EPICSName: VacLevelMaxS
    Else
       #DEVICE_PARAM_OK := FALSE; //Invalid Hash
    END_IF;
END_FUNCTION_BLOCK
FUNCTION_BLOCK "DEVTYPE_ISRC_LEBT_INTF_MPS"
{ S7_Optimized_Access := 'TRUE' }
VERSION : 1.0
   VAR_INPUT
      "MPSOK" { ExternalAccessible := 'True'; ExternalVisible := 'False'; ExternalWritable := 'False'; } : BOOL;   //EPICS Status variable: MPSOK
      "ISrcOKtoMPS" { ExternalAccessible := 'True'; ExternalVisible := 'False'; ExternalWritable := 'False'; } : BOOL;   //EPICS Status variable: ISrcOKtoMPS
   EPICSToPLCLength { ExternalAccessible := 'False'; ExternalVisible := 'False'; ExternalWritable := 'False'; } : Int;   // Length of device command register array (in words)
   EPICSToPLCDataBlockOffset { ExternalAccessible := 'False'; ExternalVisible := 'False'; ExternalWritable := 'False'; } : Int;   // Offset in EPICS->PLC comms block where this device data resides (in words)
   EPICSToPLCParametersStart { ExternalAccessible := 'False'; ExternalVisible := 'False'; ExternalWritable := 'False'; } : Int;   // The border offset between the Command and the Parameter area
   PLCToEPICSLength { ExternalAccessible := 'False'; ExternalVisible := 'False'; ExternalWritable := 'False'; } : Int;   // Length of device status register array (in words)
   PLCToEPICSDataBlockOffset { ExternalAccessible := 'False'; ExternalVisible := 'False'; ExternalWritable := 'False'; } : Int;   // Offset in PLC->EPICS comms block where this device data resides (in words)
   END_VAR
   VAR_OUTPUT
      DEVICE_PARAM_OK { ExternalAccessible := 'False'; ExternalVisible := 'False'; ExternalWritable := 'False'; } : Bool;
   END_VAR
   VAR_IN_OUT
   END_VAR
   Var DB_SPECIFIC
      MyWord { ExternalAccessible := 'False'; ExternalVisible := 'False'; ExternalWritable := 'False'; } : Word;
      MyBytesinWord { ExternalAccessible := 'False'; ExternalVisible := 'False'; ExternalWritable := 'False'; } AT MyWord : Array[0..1] of Byte;
      MyBoolsinWord { ExternalAccessible := 'False'; ExternalVisible := 'False'; ExternalWritable := 'False'; } AT MyWord : Array[0..15] of Bool;
      MyDInt { ExternalAccessible := 'False'; ExternalVisible := 'False'; ExternalWritable := 'False'; } : DInt;
      MyWordsinDint { ExternalAccessible := 'False'; ExternalVisible := 'False'; ExternalWritable := 'False'; } AT MyDInt : Array[0..1] of Word;
      MyReal { ExternalAccessible := 'False'; ExternalVisible := 'False'; ExternalWritable := 'False'; } : Real;
      MyWordsinReal { ExternalAccessible := 'False'; ExternalVisible := 'False'; ExternalWritable := 'False'; } AT MyReal : Array[0..1] of Word;
      MyInt { ExternalAccessible := 'False'; ExternalVisible := 'False'; ExternalWritable := 'False'; } : Int;
      MyWordinInt { ExternalAccessible := 'False'; ExternalVisible := 'False'; ExternalWritable := 'False'; } AT MyInt : Word;
      MyDWord { ExternalAccessible := 'False'; ExternalVisible := 'False'; ExternalWritable := 'False'; } : DWord;
      MyWordsinDWord { ExternalAccessible := 'False'; ExternalVisible := 'False'; ExternalWritable := 'False'; } AT MyDWord : Array[0..1] of Word;
      MyTime { ExternalAccessible := 'False'; ExternalVisible := 'False'; ExternalWritable := 'False'; } : Time;
      MyWordsinTime { ExternalAccessible := 'False'; ExternalVisible := 'False'; ExternalWritable := 'False'; } AT MyTime : Array[0..1] of Word;
      MyString { ExternalAccessible := 'False'; ExternalVisible := 'False'; ExternalWritable := 'False'; } : String[40];
      MyWordsinString { ExternalAccessible := 'False'; ExternalVisible := 'False'; ExternalWritable := 'False'; } AT MyString : Array[0..20] of Word;
   END_VAR
   VAR_TEMP
      HashModbus : DInt;
      HashIFA : DInt;
      HashTIAMap : DInt;
      i : Int;
   END_VAR
    //Author: Miklos Boros (miklos.boros@esss.se), Copyrigth 2017-2019 by European Spallation Source, Lund
    //This block was generated by PLCFactory, please don't change it MANUALLY!
    //Input File Name: ISrc-010_Ctrl-PLC-01-template-IFA-20191106135317.ifa
    //Generated: 20191106135317
    //According to HASH: 1347332123
    //Device type: ISRC_LEBT_INTF_MPS
    //Description: This function does the variable mapping for a device. All device-variable will be linked to an interface variable defined in this block.

    //********************************************
    //****************HASH check******************
    //********************************************


    #MyWordsinDint[0] := "EPICSToPLC"."Word"[0];
    #MyWordsinDint[1] := "EPICSToPLC"."Word"[1];
    #HashModbus := #MyDInt; //Hash from EPICS/ModbusTCP

    #HashIFA := 1347332123; //Hash from Interface Factory as a constant

    #MyWordsinDint[0] := "PLCToEPICS"."Word"[0];
    #MyWordsinDint[1] := "PLCToEPICS"."Word"[1];
    #HashTIAMap := #MyDInt; //Hash from PLCFactory TIA Map


    IF ((#HashIFA = #HashModbus) AND (#HashModbus = #HashTIAMap)) THEN //Check CRCs
        #DEVICE_PARAM_OK := TRUE;
       //###########################  ISRC_LEBT interface with MPS  ##############################
       //###########################
       //STATUS BLOCK
       //###########################

    //********************************************
    //*************STATUS VARIABLES***************
    //********************************************


       #MyWord := W#0;
       #MyBoolsinWord[8] := #"MPSOK";    //EPICSName: MPSOK
       #MyBoolsinWord[9] := #"ISrcOKtoMPS";    //EPICSName: ISrcOKtoMPS
       "PLCToEPICS"."Word"[#PLCToEPICSDataBlockOffset + 0] := #MyWord;
    Else
       #DEVICE_PARAM_OK := FALSE; //Invalid Hash
    END_IF;
END_FUNCTION_BLOCK
FUNCTION_BLOCK "DEVTYPE_ISRC_LEBT_INTF_PSS"
{ S7_Optimized_Access := 'TRUE' }
VERSION : 1.0
   VAR_INPUT
      "PSSOK" { ExternalAccessible := 'True'; ExternalVisible := 'False'; ExternalWritable := 'False'; } : BOOL;   //EPICS Status variable: PSSOK
      "HVPermitR" { ExternalAccessible := 'True'; ExternalVisible := 'False'; ExternalWritable := 'False'; } : BOOL;   //EPICS Status variable: HVPermitR
   EPICSToPLCLength { ExternalAccessible := 'False'; ExternalVisible := 'False'; ExternalWritable := 'False'; } : Int;   // Length of device command register array (in words)
   EPICSToPLCDataBlockOffset { ExternalAccessible := 'False'; ExternalVisible := 'False'; ExternalWritable := 'False'; } : Int;   // Offset in EPICS->PLC comms block where this device data resides (in words)
   EPICSToPLCParametersStart { ExternalAccessible := 'False'; ExternalVisible := 'False'; ExternalWritable := 'False'; } : Int;   // The border offset between the Command and the Parameter area
   PLCToEPICSLength { ExternalAccessible := 'False'; ExternalVisible := 'False'; ExternalWritable := 'False'; } : Int;   // Length of device status register array (in words)
   PLCToEPICSDataBlockOffset { ExternalAccessible := 'False'; ExternalVisible := 'False'; ExternalWritable := 'False'; } : Int;   // Offset in PLC->EPICS comms block where this device data resides (in words)
   END_VAR
   VAR_OUTPUT
      DEVICE_PARAM_OK { ExternalAccessible := 'False'; ExternalVisible := 'False'; ExternalWritable := 'False'; } : Bool;
   END_VAR
   VAR_IN_OUT
   END_VAR
   Var DB_SPECIFIC
      MyWord { ExternalAccessible := 'False'; ExternalVisible := 'False'; ExternalWritable := 'False'; } : Word;
      MyBytesinWord { ExternalAccessible := 'False'; ExternalVisible := 'False'; ExternalWritable := 'False'; } AT MyWord : Array[0..1] of Byte;
      MyBoolsinWord { ExternalAccessible := 'False'; ExternalVisible := 'False'; ExternalWritable := 'False'; } AT MyWord : Array[0..15] of Bool;
      MyDInt { ExternalAccessible := 'False'; ExternalVisible := 'False'; ExternalWritable := 'False'; } : DInt;
      MyWordsinDint { ExternalAccessible := 'False'; ExternalVisible := 'False'; ExternalWritable := 'False'; } AT MyDInt : Array[0..1] of Word;
      MyReal { ExternalAccessible := 'False'; ExternalVisible := 'False'; ExternalWritable := 'False'; } : Real;
      MyWordsinReal { ExternalAccessible := 'False'; ExternalVisible := 'False'; ExternalWritable := 'False'; } AT MyReal : Array[0..1] of Word;
      MyInt { ExternalAccessible := 'False'; ExternalVisible := 'False'; ExternalWritable := 'False'; } : Int;
      MyWordinInt { ExternalAccessible := 'False'; ExternalVisible := 'False'; ExternalWritable := 'False'; } AT MyInt : Word;
      MyDWord { ExternalAccessible := 'False'; ExternalVisible := 'False'; ExternalWritable := 'False'; } : DWord;
      MyWordsinDWord { ExternalAccessible := 'False'; ExternalVisible := 'False'; ExternalWritable := 'False'; } AT MyDWord : Array[0..1] of Word;
      MyTime { ExternalAccessible := 'False'; ExternalVisible := 'False'; ExternalWritable := 'False'; } : Time;
      MyWordsinTime { ExternalAccessible := 'False'; ExternalVisible := 'False'; ExternalWritable := 'False'; } AT MyTime : Array[0..1] of Word;
      MyString { ExternalAccessible := 'False'; ExternalVisible := 'False'; ExternalWritable := 'False'; } : String[40];
      MyWordsinString { ExternalAccessible := 'False'; ExternalVisible := 'False'; ExternalWritable := 'False'; } AT MyString : Array[0..20] of Word;
   END_VAR
   VAR_TEMP
      HashModbus : DInt;
      HashIFA : DInt;
      HashTIAMap : DInt;
      i : Int;
   END_VAR
    //Author: Miklos Boros (miklos.boros@esss.se), Copyrigth 2017-2019 by European Spallation Source, Lund
    //This block was generated by PLCFactory, please don't change it MANUALLY!
    //Input File Name: ISrc-010_Ctrl-PLC-01-template-IFA-20191106135317.ifa
    //Generated: 20191106135317
    //According to HASH: 1347332123
    //Device type: ISRC_LEBT_INTF_PSS
    //Description: This function does the variable mapping for a device. All device-variable will be linked to an interface variable defined in this block.

    //********************************************
    //****************HASH check******************
    //********************************************


    #MyWordsinDint[0] := "EPICSToPLC"."Word"[0];
    #MyWordsinDint[1] := "EPICSToPLC"."Word"[1];
    #HashModbus := #MyDInt; //Hash from EPICS/ModbusTCP

    #HashIFA := 1347332123; //Hash from Interface Factory as a constant

    #MyWordsinDint[0] := "PLCToEPICS"."Word"[0];
    #MyWordsinDint[1] := "PLCToEPICS"."Word"[1];
    #HashTIAMap := #MyDInt; //Hash from PLCFactory TIA Map


    IF ((#HashIFA = #HashModbus) AND (#HashModbus = #HashTIAMap)) THEN //Check CRCs
        #DEVICE_PARAM_OK := TRUE;
       //###########################  ISRC_LEBT interface with PSS  ##############################
       //###########################
       //STATUS BLOCK
       //###########################

    //********************************************
    //*************STATUS VARIABLES***************
    //********************************************


       #MyWord := W#0;
       #MyBoolsinWord[8] := #"PSSOK";    //EPICSName: PSSOK
       #MyBoolsinWord[9] := #"HVPermitR";    //EPICSName: HVPermitR
       "PLCToEPICS"."Word"[#PLCToEPICSDataBlockOffset + 0] := #MyWord;
    Else
       #DEVICE_PARAM_OK := FALSE; //Invalid Hash
    END_IF;
END_FUNCTION_BLOCK
FUNCTION_BLOCK "DEVTYPE_ISRC_LEBT_INTF_VAC"
{ S7_Optimized_Access := 'TRUE' }
VERSION : 1.0
   VAR_INPUT
      "VacOK" { ExternalAccessible := 'True'; ExternalVisible := 'False'; ExternalWritable := 'False'; } : BOOL;   //EPICS Status variable: VacOK
      "VacPermit" { ExternalAccessible := 'True'; ExternalVisible := 'False'; ExternalWritable := 'False'; } : BOOL;   //EPICS Status variable: VacPermit
   EPICSToPLCLength { ExternalAccessible := 'False'; ExternalVisible := 'False'; ExternalWritable := 'False'; } : Int;   // Length of device command register array (in words)
   EPICSToPLCDataBlockOffset { ExternalAccessible := 'False'; ExternalVisible := 'False'; ExternalWritable := 'False'; } : Int;   // Offset in EPICS->PLC comms block where this device data resides (in words)
   EPICSToPLCParametersStart { ExternalAccessible := 'False'; ExternalVisible := 'False'; ExternalWritable := 'False'; } : Int;   // The border offset between the Command and the Parameter area
   PLCToEPICSLength { ExternalAccessible := 'False'; ExternalVisible := 'False'; ExternalWritable := 'False'; } : Int;   // Length of device status register array (in words)
   PLCToEPICSDataBlockOffset { ExternalAccessible := 'False'; ExternalVisible := 'False'; ExternalWritable := 'False'; } : Int;   // Offset in PLC->EPICS comms block where this device data resides (in words)
   END_VAR
   VAR_OUTPUT
      DEVICE_PARAM_OK { ExternalAccessible := 'False'; ExternalVisible := 'False'; ExternalWritable := 'False'; } : Bool;
   END_VAR
   VAR_IN_OUT
   END_VAR
   Var DB_SPECIFIC
      MyWord { ExternalAccessible := 'False'; ExternalVisible := 'False'; ExternalWritable := 'False'; } : Word;
      MyBytesinWord { ExternalAccessible := 'False'; ExternalVisible := 'False'; ExternalWritable := 'False'; } AT MyWord : Array[0..1] of Byte;
      MyBoolsinWord { ExternalAccessible := 'False'; ExternalVisible := 'False'; ExternalWritable := 'False'; } AT MyWord : Array[0..15] of Bool;
      MyDInt { ExternalAccessible := 'False'; ExternalVisible := 'False'; ExternalWritable := 'False'; } : DInt;
      MyWordsinDint { ExternalAccessible := 'False'; ExternalVisible := 'False'; ExternalWritable := 'False'; } AT MyDInt : Array[0..1] of Word;
      MyReal { ExternalAccessible := 'False'; ExternalVisible := 'False'; ExternalWritable := 'False'; } : Real;
      MyWordsinReal { ExternalAccessible := 'False'; ExternalVisible := 'False'; ExternalWritable := 'False'; } AT MyReal : Array[0..1] of Word;
      MyInt { ExternalAccessible := 'False'; ExternalVisible := 'False'; ExternalWritable := 'False'; } : Int;
      MyWordinInt { ExternalAccessible := 'False'; ExternalVisible := 'False'; ExternalWritable := 'False'; } AT MyInt : Word;
      MyDWord { ExternalAccessible := 'False'; ExternalVisible := 'False'; ExternalWritable := 'False'; } : DWord;
      MyWordsinDWord { ExternalAccessible := 'False'; ExternalVisible := 'False'; ExternalWritable := 'False'; } AT MyDWord : Array[0..1] of Word;
      MyTime { ExternalAccessible := 'False'; ExternalVisible := 'False'; ExternalWritable := 'False'; } : Time;
      MyWordsinTime { ExternalAccessible := 'False'; ExternalVisible := 'False'; ExternalWritable := 'False'; } AT MyTime : Array[0..1] of Word;
      MyString { ExternalAccessible := 'False'; ExternalVisible := 'False'; ExternalWritable := 'False'; } : String[40];
      MyWordsinString { ExternalAccessible := 'False'; ExternalVisible := 'False'; ExternalWritable := 'False'; } AT MyString : Array[0..20] of Word;
   END_VAR
   VAR_TEMP
      HashModbus : DInt;
      HashIFA : DInt;
      HashTIAMap : DInt;
      i : Int;
   END_VAR
    //Author: Miklos Boros (miklos.boros@esss.se), Copyrigth 2017-2019 by European Spallation Source, Lund
    //This block was generated by PLCFactory, please don't change it MANUALLY!
    //Input File Name: ISrc-010_Ctrl-PLC-01-template-IFA-20191106135317.ifa
    //Generated: 20191106135317
    //According to HASH: 1347332123
    //Device type: ISRC_LEBT_INTF_VAC
    //Description: This function does the variable mapping for a device. All device-variable will be linked to an interface variable defined in this block.

    //********************************************
    //****************HASH check******************
    //********************************************


    #MyWordsinDint[0] := "EPICSToPLC"."Word"[0];
    #MyWordsinDint[1] := "EPICSToPLC"."Word"[1];
    #HashModbus := #MyDInt; //Hash from EPICS/ModbusTCP

    #HashIFA := 1347332123; //Hash from Interface Factory as a constant

    #MyWordsinDint[0] := "PLCToEPICS"."Word"[0];
    #MyWordsinDint[1] := "PLCToEPICS"."Word"[1];
    #HashTIAMap := #MyDInt; //Hash from PLCFactory TIA Map


    IF ((#HashIFA = #HashModbus) AND (#HashModbus = #HashTIAMap)) THEN //Check CRCs
        #DEVICE_PARAM_OK := TRUE;
       //###########################  ISRC_LEBT interface with Vacuum System  ##############################
       //###########################
       //STATUS BLOCK
       //###########################

    //********************************************
    //*************STATUS VARIABLES***************
    //********************************************


       #MyWord := W#0;
       #MyBoolsinWord[8] := #"VacOK";    //EPICSName: VacOK
       #MyBoolsinWord[9] := #"VacPermit";    //EPICSName: VacPermit
       "PLCToEPICS"."Word"[#PLCToEPICSDataBlockOffset + 0] := #MyWord;
    Else
       #DEVICE_PARAM_OK := FALSE; //Invalid Hash
    END_IF;
END_FUNCTION_BLOCK
FUNCTION_BLOCK "DEVTYPE_ISRC_LEBT_IRIS"
{ S7_Optimized_Access := 'TRUE' }
VERSION : 1.0
   VAR_INPUT
      "WtrFlowOK" { ExternalAccessible := 'True'; ExternalVisible := 'False'; ExternalWritable := 'False'; } : BOOL;   //EPICS Status variable: WtrFlowOK
      "WtrTempMax1Err" { ExternalAccessible := 'True'; ExternalVisible := 'False'; ExternalWritable := 'False'; } : BOOL;   //EPICS Status variable: WtrTempMax1Err
      "WtrTempMax2Err" { ExternalAccessible := 'True'; ExternalVisible := 'False'; ExternalWritable := 'False'; } : BOOL;   //EPICS Status variable: WtrTempMax2Err
   EPICSToPLCLength { ExternalAccessible := 'False'; ExternalVisible := 'False'; ExternalWritable := 'False'; } : Int;   // Length of device command register array (in words)
   EPICSToPLCDataBlockOffset { ExternalAccessible := 'False'; ExternalVisible := 'False'; ExternalWritable := 'False'; } : Int;   // Offset in EPICS->PLC comms block where this device data resides (in words)
   EPICSToPLCParametersStart { ExternalAccessible := 'False'; ExternalVisible := 'False'; ExternalWritable := 'False'; } : Int;   // The border offset between the Command and the Parameter area
   PLCToEPICSLength { ExternalAccessible := 'False'; ExternalVisible := 'False'; ExternalWritable := 'False'; } : Int;   // Length of device status register array (in words)
   PLCToEPICSDataBlockOffset { ExternalAccessible := 'False'; ExternalVisible := 'False'; ExternalWritable := 'False'; } : Int;   // Offset in PLC->EPICS comms block where this device data resides (in words)
   END_VAR
   VAR_OUTPUT
      DEVICE_PARAM_OK { ExternalAccessible := 'False'; ExternalVisible := 'False'; ExternalWritable := 'False'; } : Bool;
   END_VAR
   VAR_IN_OUT
   END_VAR
   Var DB_SPECIFIC
      MyWord { ExternalAccessible := 'False'; ExternalVisible := 'False'; ExternalWritable := 'False'; } : Word;
      MyBytesinWord { ExternalAccessible := 'False'; ExternalVisible := 'False'; ExternalWritable := 'False'; } AT MyWord : Array[0..1] of Byte;
      MyBoolsinWord { ExternalAccessible := 'False'; ExternalVisible := 'False'; ExternalWritable := 'False'; } AT MyWord : Array[0..15] of Bool;
      MyDInt { ExternalAccessible := 'False'; ExternalVisible := 'False'; ExternalWritable := 'False'; } : DInt;
      MyWordsinDint { ExternalAccessible := 'False'; ExternalVisible := 'False'; ExternalWritable := 'False'; } AT MyDInt : Array[0..1] of Word;
      MyReal { ExternalAccessible := 'False'; ExternalVisible := 'False'; ExternalWritable := 'False'; } : Real;
      MyWordsinReal { ExternalAccessible := 'False'; ExternalVisible := 'False'; ExternalWritable := 'False'; } AT MyReal : Array[0..1] of Word;
      MyInt { ExternalAccessible := 'False'; ExternalVisible := 'False'; ExternalWritable := 'False'; } : Int;
      MyWordinInt { ExternalAccessible := 'False'; ExternalVisible := 'False'; ExternalWritable := 'False'; } AT MyInt : Word;
      MyDWord { ExternalAccessible := 'False'; ExternalVisible := 'False'; ExternalWritable := 'False'; } : DWord;
      MyWordsinDWord { ExternalAccessible := 'False'; ExternalVisible := 'False'; ExternalWritable := 'False'; } AT MyDWord : Array[0..1] of Word;
      MyTime { ExternalAccessible := 'False'; ExternalVisible := 'False'; ExternalWritable := 'False'; } : Time;
      MyWordsinTime { ExternalAccessible := 'False'; ExternalVisible := 'False'; ExternalWritable := 'False'; } AT MyTime : Array[0..1] of Word;
      MyString { ExternalAccessible := 'False'; ExternalVisible := 'False'; ExternalWritable := 'False'; } : String[40];
      MyWordsinString { ExternalAccessible := 'False'; ExternalVisible := 'False'; ExternalWritable := 'False'; } AT MyString : Array[0..20] of Word;
   END_VAR
   VAR_TEMP
      HashModbus : DInt;
      HashIFA : DInt;
      HashTIAMap : DInt;
      i : Int;
   END_VAR
    //Author: Miklos Boros (miklos.boros@esss.se), Copyrigth 2017-2019 by European Spallation Source, Lund
    //This block was generated by PLCFactory, please don't change it MANUALLY!
    //Input File Name: ISrc-010_Ctrl-PLC-01-template-IFA-20191106135317.ifa
    //Generated: 20191106135317
    //According to HASH: 1347332123
    //Device type: ISRC_LEBT_IRIS
    //Description: This function does the variable mapping for a device. All device-variable will be linked to an interface variable defined in this block.

    //********************************************
    //****************HASH check******************
    //********************************************


    #MyWordsinDint[0] := "EPICSToPLC"."Word"[0];
    #MyWordsinDint[1] := "EPICSToPLC"."Word"[1];
    #HashModbus := #MyDInt; //Hash from EPICS/ModbusTCP

    #HashIFA := 1347332123; //Hash from Interface Factory as a constant

    #MyWordsinDint[0] := "PLCToEPICS"."Word"[0];
    #MyWordsinDint[1] := "PLCToEPICS"."Word"[1];
    #HashTIAMap := #MyDInt; //Hash from PLCFactory TIA Map


    IF ((#HashIFA = #HashModbus) AND (#HashModbus = #HashTIAMap)) THEN //Check CRCs
        #DEVICE_PARAM_OK := TRUE;
       //###########################  LEBT Iris  ##############################
       //###########################
       //STATUS BLOCK
       //###########################

    //********************************************
    //*************STATUS VARIABLES***************
    //********************************************


       #MyWord := W#0;
       #MyBoolsinWord[8] := #"WtrFlowOK";    //EPICSName: WtrFlowOK
       #MyBoolsinWord[9] := #"WtrTempMax1Err";    //EPICSName: WtrTempMax1Err
       #MyBoolsinWord[10] := #"WtrTempMax2Err";    //EPICSName: WtrTempMax2Err
       "PLCToEPICS"."Word"[#PLCToEPICSDataBlockOffset + 0] := #MyWord;
    Else
       #DEVICE_PARAM_OK := FALSE; //Invalid Hash
    END_IF;
END_FUNCTION_BLOCK
FUNCTION_BLOCK "DEVTYPE_ISRC_LEBT_Magtr"
{ S7_Optimized_Access := 'TRUE' }
VERSION : 1.0
   VAR_INPUT
      "EnCmdR" { ExternalAccessible := 'True'; ExternalVisible := 'False'; ExternalWritable := 'False'; } : BOOL;   //EPICS Status variable: EnCmdR
      "MWPowerOnR" { ExternalAccessible := 'True'; ExternalVisible := 'False'; ExternalWritable := 'False'; } : BOOL;   //EPICS Status variable: MWPowerOnR
      "PulseModeOK" { ExternalAccessible := 'True'; ExternalVisible := 'False'; ExternalWritable := 'False'; } : BOOL;   //EPICS Status variable: PulseModeOK
   EPICSToPLCLength { ExternalAccessible := 'False'; ExternalVisible := 'False'; ExternalWritable := 'False'; } : Int;   // Length of device command register array (in words)
   EPICSToPLCDataBlockOffset { ExternalAccessible := 'False'; ExternalVisible := 'False'; ExternalWritable := 'False'; } : Int;   // Offset in EPICS->PLC comms block where this device data resides (in words)
   EPICSToPLCParametersStart { ExternalAccessible := 'False'; ExternalVisible := 'False'; ExternalWritable := 'False'; } : Int;   // The border offset between the Command and the Parameter area
   PLCToEPICSLength { ExternalAccessible := 'False'; ExternalVisible := 'False'; ExternalWritable := 'False'; } : Int;   // Length of device status register array (in words)
   PLCToEPICSDataBlockOffset { ExternalAccessible := 'False'; ExternalVisible := 'False'; ExternalWritable := 'False'; } : Int;   // Offset in PLC->EPICS comms block where this device data resides (in words)
   END_VAR
   VAR_OUTPUT
      "iPulseMode" { ExternalAccessible := 'True'; ExternalVisible := 'False'; ExternalWritable := 'False'; } : BOOL;   //EPICS Parameter variable: iPulseMode
      DEVICE_PARAM_OK { ExternalAccessible := 'False'; ExternalVisible := 'False'; ExternalWritable := 'False'; } : Bool;
   END_VAR
   VAR_IN_OUT
   END_VAR
   Var DB_SPECIFIC
      MyWord { ExternalAccessible := 'False'; ExternalVisible := 'False'; ExternalWritable := 'False'; } : Word;
      MyBytesinWord { ExternalAccessible := 'False'; ExternalVisible := 'False'; ExternalWritable := 'False'; } AT MyWord : Array[0..1] of Byte;
      MyBoolsinWord { ExternalAccessible := 'False'; ExternalVisible := 'False'; ExternalWritable := 'False'; } AT MyWord : Array[0..15] of Bool;
      MyDInt { ExternalAccessible := 'False'; ExternalVisible := 'False'; ExternalWritable := 'False'; } : DInt;
      MyWordsinDint { ExternalAccessible := 'False'; ExternalVisible := 'False'; ExternalWritable := 'False'; } AT MyDInt : Array[0..1] of Word;
      MyReal { ExternalAccessible := 'False'; ExternalVisible := 'False'; ExternalWritable := 'False'; } : Real;
      MyWordsinReal { ExternalAccessible := 'False'; ExternalVisible := 'False'; ExternalWritable := 'False'; } AT MyReal : Array[0..1] of Word;
      MyInt { ExternalAccessible := 'False'; ExternalVisible := 'False'; ExternalWritable := 'False'; } : Int;
      MyWordinInt { ExternalAccessible := 'False'; ExternalVisible := 'False'; ExternalWritable := 'False'; } AT MyInt : Word;
      MyDWord { ExternalAccessible := 'False'; ExternalVisible := 'False'; ExternalWritable := 'False'; } : DWord;
      MyWordsinDWord { ExternalAccessible := 'False'; ExternalVisible := 'False'; ExternalWritable := 'False'; } AT MyDWord : Array[0..1] of Word;
      MyTime { ExternalAccessible := 'False'; ExternalVisible := 'False'; ExternalWritable := 'False'; } : Time;
      MyWordsinTime { ExternalAccessible := 'False'; ExternalVisible := 'False'; ExternalWritable := 'False'; } AT MyTime : Array[0..1] of Word;
      MyString { ExternalAccessible := 'False'; ExternalVisible := 'False'; ExternalWritable := 'False'; } : String[40];
      MyWordsinString { ExternalAccessible := 'False'; ExternalVisible := 'False'; ExternalWritable := 'False'; } AT MyString : Array[0..20] of Word;
   END_VAR
   VAR_TEMP
      HashModbus : DInt;
      HashIFA : DInt;
      HashTIAMap : DInt;
      i : Int;
   END_VAR
    //Author: Miklos Boros (miklos.boros@esss.se), Copyrigth 2017-2019 by European Spallation Source, Lund
    //This block was generated by PLCFactory, please don't change it MANUALLY!
    //Input File Name: ISrc-010_Ctrl-PLC-01-template-IFA-20191106135317.ifa
    //Generated: 20191106135317
    //According to HASH: 1347332123
    //Device type: ISRC_LEBT_Magtr
    //Description: This function does the variable mapping for a device. All device-variable will be linked to an interface variable defined in this block.

    //********************************************
    //****************HASH check******************
    //********************************************


    #MyWordsinDint[0] := "EPICSToPLC"."Word"[0];
    #MyWordsinDint[1] := "EPICSToPLC"."Word"[1];
    #HashModbus := #MyDInt; //Hash from EPICS/ModbusTCP

    #HashIFA := 1347332123; //Hash from Interface Factory as a constant

    #MyWordsinDint[0] := "PLCToEPICS"."Word"[0];
    #MyWordsinDint[1] := "PLCToEPICS"."Word"[1];
    #HashTIAMap := #MyDInt; //Hash from PLCFactory TIA Map


    IF ((#HashIFA = #HashModbus) AND (#HashModbus = #HashTIAMap)) THEN //Check CRCs
        #DEVICE_PARAM_OK := TRUE;
       //###########################  ISRC Magnetron  ##############################
       //###########################
       //STATUS BLOCK
       //###########################

    //********************************************
    //*************STATUS VARIABLES***************
    //********************************************


       #MyWord := W#0;
       #MyBoolsinWord[8] := #"EnCmdR";    //EPICSName: EnCmdR
       #MyBoolsinWord[9] := #"MWPowerOnR";    //EPICSName: MWPowerOnR
       #MyBoolsinWord[10] := #"PulseModeOK";    //EPICSName: PulseModeOK
       "PLCToEPICS"."Word"[#PLCToEPICSDataBlockOffset + 0] := #MyWord;

    //********************************************
    //************PARAMETER VARIABLES*************
    //********************************************


       #MyWord := "EPICSToPLC"."Word"[#EPICSToPLCDataBlockOffset + 0];
       #"iPulseMode" := #MyBoolsinWord[8];    //EPICSName: iPulseMode
    Else
       #DEVICE_PARAM_OK := FALSE; //Invalid Hash
    END_IF;
END_FUNCTION_BLOCK
FUNCTION_BLOCK "DEVTYPE_ISRC_LEBT_MatTr"
{ S7_Optimized_Access := 'TRUE' }
VERSION : 1.0
   VAR_INPUT
      "WtrFlowOK" { ExternalAccessible := 'True'; ExternalVisible := 'False'; ExternalWritable := 'False'; } : BOOL;   //EPICS Status variable: WtrFlowOK
   EPICSToPLCLength { ExternalAccessible := 'False'; ExternalVisible := 'False'; ExternalWritable := 'False'; } : Int;   // Length of device command register array (in words)
   EPICSToPLCDataBlockOffset { ExternalAccessible := 'False'; ExternalVisible := 'False'; ExternalWritable := 'False'; } : Int;   // Offset in EPICS->PLC comms block where this device data resides (in words)
   EPICSToPLCParametersStart { ExternalAccessible := 'False'; ExternalVisible := 'False'; ExternalWritable := 'False'; } : Int;   // The border offset between the Command and the Parameter area
   PLCToEPICSLength { ExternalAccessible := 'False'; ExternalVisible := 'False'; ExternalWritable := 'False'; } : Int;   // Length of device status register array (in words)
   PLCToEPICSDataBlockOffset { ExternalAccessible := 'False'; ExternalVisible := 'False'; ExternalWritable := 'False'; } : Int;   // Offset in PLC->EPICS comms block where this device data resides (in words)
   END_VAR
   VAR_OUTPUT
      DEVICE_PARAM_OK { ExternalAccessible := 'False'; ExternalVisible := 'False'; ExternalWritable := 'False'; } : Bool;
   END_VAR
   VAR_IN_OUT
   END_VAR
   Var DB_SPECIFIC
      MyWord { ExternalAccessible := 'False'; ExternalVisible := 'False'; ExternalWritable := 'False'; } : Word;
      MyBytesinWord { ExternalAccessible := 'False'; ExternalVisible := 'False'; ExternalWritable := 'False'; } AT MyWord : Array[0..1] of Byte;
      MyBoolsinWord { ExternalAccessible := 'False'; ExternalVisible := 'False'; ExternalWritable := 'False'; } AT MyWord : Array[0..15] of Bool;
      MyDInt { ExternalAccessible := 'False'; ExternalVisible := 'False'; ExternalWritable := 'False'; } : DInt;
      MyWordsinDint { ExternalAccessible := 'False'; ExternalVisible := 'False'; ExternalWritable := 'False'; } AT MyDInt : Array[0..1] of Word;
      MyReal { ExternalAccessible := 'False'; ExternalVisible := 'False'; ExternalWritable := 'False'; } : Real;
      MyWordsinReal { ExternalAccessible := 'False'; ExternalVisible := 'False'; ExternalWritable := 'False'; } AT MyReal : Array[0..1] of Word;
      MyInt { ExternalAccessible := 'False'; ExternalVisible := 'False'; ExternalWritable := 'False'; } : Int;
      MyWordinInt { ExternalAccessible := 'False'; ExternalVisible := 'False'; ExternalWritable := 'False'; } AT MyInt : Word;
      MyDWord { ExternalAccessible := 'False'; ExternalVisible := 'False'; ExternalWritable := 'False'; } : DWord;
      MyWordsinDWord { ExternalAccessible := 'False'; ExternalVisible := 'False'; ExternalWritable := 'False'; } AT MyDWord : Array[0..1] of Word;
      MyTime { ExternalAccessible := 'False'; ExternalVisible := 'False'; ExternalWritable := 'False'; } : Time;
      MyWordsinTime { ExternalAccessible := 'False'; ExternalVisible := 'False'; ExternalWritable := 'False'; } AT MyTime : Array[0..1] of Word;
      MyString { ExternalAccessible := 'False'; ExternalVisible := 'False'; ExternalWritable := 'False'; } : String[40];
      MyWordsinString { ExternalAccessible := 'False'; ExternalVisible := 'False'; ExternalWritable := 'False'; } AT MyString : Array[0..20] of Word;
   END_VAR
   VAR_TEMP
      HashModbus : DInt;
      HashIFA : DInt;
      HashTIAMap : DInt;
      i : Int;
   END_VAR
    //Author: Miklos Boros (miklos.boros@esss.se), Copyrigth 2017-2019 by European Spallation Source, Lund
    //This block was generated by PLCFactory, please don't change it MANUALLY!
    //Input File Name: ISrc-010_Ctrl-PLC-01-template-IFA-20191106135317.ifa
    //Generated: 20191106135317
    //According to HASH: 1347332123
    //Device type: ISRC_LEBT_MatTr
    //Description: This function does the variable mapping for a device. All device-variable will be linked to an interface variable defined in this block.

    //********************************************
    //****************HASH check******************
    //********************************************


    #MyWordsinDint[0] := "EPICSToPLC"."Word"[0];
    #MyWordsinDint[1] := "EPICSToPLC"."Word"[1];
    #HashModbus := #MyDInt; //Hash from EPICS/ModbusTCP

    #HashIFA := 1347332123; //Hash from Interface Factory as a constant

    #MyWordsinDint[0] := "PLCToEPICS"."Word"[0];
    #MyWordsinDint[1] := "PLCToEPICS"."Word"[1];
    #HashTIAMap := #MyDInt; //Hash from PLCFactory TIA Map


    IF ((#HashIFA = #HashModbus) AND (#HashModbus = #HashTIAMap)) THEN //Check CRCs
        #DEVICE_PARAM_OK := TRUE;
       //###########################  ISRC_LEBT Matching Transformer  ##############################
       //###########################
       //STATUS BLOCK
       //###########################

    //********************************************
    //*************STATUS VARIABLES***************
    //********************************************


       #MyWord := W#0;
       #MyBoolsinWord[8] := #"WtrFlowOK";    //EPICSName: WtrFlowOK
       "PLCToEPICS"."Word"[#PLCToEPICSDataBlockOffset + 0] := #MyWord;
    Else
       #DEVICE_PARAM_OK := FALSE; //Invalid Hash
    END_IF;
END_FUNCTION_BLOCK
FUNCTION_BLOCK "DEVTYPE_ISRC_LEBT_PBI_EMU"
{ S7_Optimized_Access := 'TRUE' }
VERSION : 1.0
   VAR_INPUT
      "HorWtrFlowOK" { ExternalAccessible := 'True'; ExternalVisible := 'False'; ExternalWritable := 'False'; } : BOOL;   //EPICS Status variable: HorWtrFlowOK
      "VerWtrFlowOK" { ExternalAccessible := 'True'; ExternalVisible := 'False'; ExternalWritable := 'False'; } : BOOL;   //EPICS Status variable: VerWtrFlowOK
   EPICSToPLCLength { ExternalAccessible := 'False'; ExternalVisible := 'False'; ExternalWritable := 'False'; } : Int;   // Length of device command register array (in words)
   EPICSToPLCDataBlockOffset { ExternalAccessible := 'False'; ExternalVisible := 'False'; ExternalWritable := 'False'; } : Int;   // Offset in EPICS->PLC comms block where this device data resides (in words)
   EPICSToPLCParametersStart { ExternalAccessible := 'False'; ExternalVisible := 'False'; ExternalWritable := 'False'; } : Int;   // The border offset between the Command and the Parameter area
   PLCToEPICSLength { ExternalAccessible := 'False'; ExternalVisible := 'False'; ExternalWritable := 'False'; } : Int;   // Length of device status register array (in words)
   PLCToEPICSDataBlockOffset { ExternalAccessible := 'False'; ExternalVisible := 'False'; ExternalWritable := 'False'; } : Int;   // Offset in PLC->EPICS comms block where this device data resides (in words)
   END_VAR
   VAR_OUTPUT
      DEVICE_PARAM_OK { ExternalAccessible := 'False'; ExternalVisible := 'False'; ExternalWritable := 'False'; } : Bool;
   END_VAR
   VAR_IN_OUT
   END_VAR
   Var DB_SPECIFIC
      MyWord { ExternalAccessible := 'False'; ExternalVisible := 'False'; ExternalWritable := 'False'; } : Word;
      MyBytesinWord { ExternalAccessible := 'False'; ExternalVisible := 'False'; ExternalWritable := 'False'; } AT MyWord : Array[0..1] of Byte;
      MyBoolsinWord { ExternalAccessible := 'False'; ExternalVisible := 'False'; ExternalWritable := 'False'; } AT MyWord : Array[0..15] of Bool;
      MyDInt { ExternalAccessible := 'False'; ExternalVisible := 'False'; ExternalWritable := 'False'; } : DInt;
      MyWordsinDint { ExternalAccessible := 'False'; ExternalVisible := 'False'; ExternalWritable := 'False'; } AT MyDInt : Array[0..1] of Word;
      MyReal { ExternalAccessible := 'False'; ExternalVisible := 'False'; ExternalWritable := 'False'; } : Real;
      MyWordsinReal { ExternalAccessible := 'False'; ExternalVisible := 'False'; ExternalWritable := 'False'; } AT MyReal : Array[0..1] of Word;
      MyInt { ExternalAccessible := 'False'; ExternalVisible := 'False'; ExternalWritable := 'False'; } : Int;
      MyWordinInt { ExternalAccessible := 'False'; ExternalVisible := 'False'; ExternalWritable := 'False'; } AT MyInt : Word;
      MyDWord { ExternalAccessible := 'False'; ExternalVisible := 'False'; ExternalWritable := 'False'; } : DWord;
      MyWordsinDWord { ExternalAccessible := 'False'; ExternalVisible := 'False'; ExternalWritable := 'False'; } AT MyDWord : Array[0..1] of Word;
      MyTime { ExternalAccessible := 'False'; ExternalVisible := 'False'; ExternalWritable := 'False'; } : Time;
      MyWordsinTime { ExternalAccessible := 'False'; ExternalVisible := 'False'; ExternalWritable := 'False'; } AT MyTime : Array[0..1] of Word;
      MyString { ExternalAccessible := 'False'; ExternalVisible := 'False'; ExternalWritable := 'False'; } : String[40];
      MyWordsinString { ExternalAccessible := 'False'; ExternalVisible := 'False'; ExternalWritable := 'False'; } AT MyString : Array[0..20] of Word;
   END_VAR
   VAR_TEMP
      HashModbus : DInt;
      HashIFA : DInt;
      HashTIAMap : DInt;
      i : Int;
   END_VAR
    //Author: Miklos Boros (miklos.boros@esss.se), Copyrigth 2017-2019 by European Spallation Source, Lund
    //This block was generated by PLCFactory, please don't change it MANUALLY!
    //Input File Name: ISrc-010_Ctrl-PLC-01-template-IFA-20191106135317.ifa
    //Generated: 20191106135317
    //According to HASH: 1347332123
    //Device type: ISRC_LEBT_PBI_EMU
    //Description: This function does the variable mapping for a device. All device-variable will be linked to an interface variable defined in this block.

    //********************************************
    //****************HASH check******************
    //********************************************


    #MyWordsinDint[0] := "EPICSToPLC"."Word"[0];
    #MyWordsinDint[1] := "EPICSToPLC"."Word"[1];
    #HashModbus := #MyDInt; //Hash from EPICS/ModbusTCP

    #HashIFA := 1347332123; //Hash from Interface Factory as a constant

    #MyWordsinDint[0] := "PLCToEPICS"."Word"[0];
    #MyWordsinDint[1] := "PLCToEPICS"."Word"[1];
    #HashTIAMap := #MyDInt; //Hash from PLCFactory TIA Map


    IF ((#HashIFA = #HashModbus) AND (#HashModbus = #HashTIAMap)) THEN //Check CRCs
        #DEVICE_PARAM_OK := TRUE;
       //###########################  LEBT EMU  ##############################
       //###########################
       //STATUS BLOCK
       //###########################

    //********************************************
    //*************STATUS VARIABLES***************
    //********************************************


       #MyWord := W#0;
       #MyBoolsinWord[8] := #"HorWtrFlowOK";    //EPICSName: HorWtrFlowOK
       #MyBoolsinWord[9] := #"VerWtrFlowOK";    //EPICSName: VerWtrFlowOK
       "PLCToEPICS"."Word"[#PLCToEPICSDataBlockOffset + 0] := #MyWord;
    Else
       #DEVICE_PARAM_OK := FALSE; //Invalid Hash
    END_IF;
END_FUNCTION_BLOCK
FUNCTION_BLOCK "DEVTYPE_ISRC_LEBT_PBI_FC"
{ S7_Optimized_Access := 'TRUE' }
VERSION : 1.0
   VAR_INPUT
      "WtrFlowOK" { ExternalAccessible := 'True'; ExternalVisible := 'False'; ExternalWritable := 'False'; } : BOOL;   //EPICS Status variable: WtrFlowOK
   EPICSToPLCLength { ExternalAccessible := 'False'; ExternalVisible := 'False'; ExternalWritable := 'False'; } : Int;   // Length of device command register array (in words)
   EPICSToPLCDataBlockOffset { ExternalAccessible := 'False'; ExternalVisible := 'False'; ExternalWritable := 'False'; } : Int;   // Offset in EPICS->PLC comms block where this device data resides (in words)
   EPICSToPLCParametersStart { ExternalAccessible := 'False'; ExternalVisible := 'False'; ExternalWritable := 'False'; } : Int;   // The border offset between the Command and the Parameter area
   PLCToEPICSLength { ExternalAccessible := 'False'; ExternalVisible := 'False'; ExternalWritable := 'False'; } : Int;   // Length of device status register array (in words)
   PLCToEPICSDataBlockOffset { ExternalAccessible := 'False'; ExternalVisible := 'False'; ExternalWritable := 'False'; } : Int;   // Offset in PLC->EPICS comms block where this device data resides (in words)
   END_VAR
   VAR_OUTPUT
      DEVICE_PARAM_OK { ExternalAccessible := 'False'; ExternalVisible := 'False'; ExternalWritable := 'False'; } : Bool;
   END_VAR
   VAR_IN_OUT
   END_VAR
   Var DB_SPECIFIC
      MyWord { ExternalAccessible := 'False'; ExternalVisible := 'False'; ExternalWritable := 'False'; } : Word;
      MyBytesinWord { ExternalAccessible := 'False'; ExternalVisible := 'False'; ExternalWritable := 'False'; } AT MyWord : Array[0..1] of Byte;
      MyBoolsinWord { ExternalAccessible := 'False'; ExternalVisible := 'False'; ExternalWritable := 'False'; } AT MyWord : Array[0..15] of Bool;
      MyDInt { ExternalAccessible := 'False'; ExternalVisible := 'False'; ExternalWritable := 'False'; } : DInt;
      MyWordsinDint { ExternalAccessible := 'False'; ExternalVisible := 'False'; ExternalWritable := 'False'; } AT MyDInt : Array[0..1] of Word;
      MyReal { ExternalAccessible := 'False'; ExternalVisible := 'False'; ExternalWritable := 'False'; } : Real;
      MyWordsinReal { ExternalAccessible := 'False'; ExternalVisible := 'False'; ExternalWritable := 'False'; } AT MyReal : Array[0..1] of Word;
      MyInt { ExternalAccessible := 'False'; ExternalVisible := 'False'; ExternalWritable := 'False'; } : Int;
      MyWordinInt { ExternalAccessible := 'False'; ExternalVisible := 'False'; ExternalWritable := 'False'; } AT MyInt : Word;
      MyDWord { ExternalAccessible := 'False'; ExternalVisible := 'False'; ExternalWritable := 'False'; } : DWord;
      MyWordsinDWord { ExternalAccessible := 'False'; ExternalVisible := 'False'; ExternalWritable := 'False'; } AT MyDWord : Array[0..1] of Word;
      MyTime { ExternalAccessible := 'False'; ExternalVisible := 'False'; ExternalWritable := 'False'; } : Time;
      MyWordsinTime { ExternalAccessible := 'False'; ExternalVisible := 'False'; ExternalWritable := 'False'; } AT MyTime : Array[0..1] of Word;
      MyString { ExternalAccessible := 'False'; ExternalVisible := 'False'; ExternalWritable := 'False'; } : String[40];
      MyWordsinString { ExternalAccessible := 'False'; ExternalVisible := 'False'; ExternalWritable := 'False'; } AT MyString : Array[0..20] of Word;
   END_VAR
   VAR_TEMP
      HashModbus : DInt;
      HashIFA : DInt;
      HashTIAMap : DInt;
      i : Int;
   END_VAR
    //Author: Miklos Boros (miklos.boros@esss.se), Copyrigth 2017-2019 by European Spallation Source, Lund
    //This block was generated by PLCFactory, please don't change it MANUALLY!
    //Input File Name: ISrc-010_Ctrl-PLC-01-template-IFA-20191106135317.ifa
    //Generated: 20191106135317
    //According to HASH: 1347332123
    //Device type: ISRC_LEBT_PBI_FC
    //Description: This function does the variable mapping for a device. All device-variable will be linked to an interface variable defined in this block.

    //********************************************
    //****************HASH check******************
    //********************************************


    #MyWordsinDint[0] := "EPICSToPLC"."Word"[0];
    #MyWordsinDint[1] := "EPICSToPLC"."Word"[1];
    #HashModbus := #MyDInt; //Hash from EPICS/ModbusTCP

    #HashIFA := 1347332123; //Hash from Interface Factory as a constant

    #MyWordsinDint[0] := "PLCToEPICS"."Word"[0];
    #MyWordsinDint[1] := "PLCToEPICS"."Word"[1];
    #HashTIAMap := #MyDInt; //Hash from PLCFactory TIA Map


    IF ((#HashIFA = #HashModbus) AND (#HashModbus = #HashTIAMap)) THEN //Check CRCs
        #DEVICE_PARAM_OK := TRUE;
       //###########################  LEBT FaradayCup  ##############################
       //###########################
       //STATUS BLOCK
       //###########################

    //********************************************
    //*************STATUS VARIABLES***************
    //********************************************


       #MyWord := W#0;
       #MyBoolsinWord[8] := #"WtrFlowOK";    //EPICSName: WtrFlowOK
       "PLCToEPICS"."Word"[#PLCToEPICSDataBlockOffset + 0] := #MyWord;
    Else
       #DEVICE_PARAM_OK := FALSE; //Invalid Hash
    END_IF;
END_FUNCTION_BLOCK
FUNCTION_BLOCK "DEVTYPE_ISRC_LEBT_PS_COIL"
{ S7_Optimized_Access := 'TRUE' }
VERSION : 1.0
   VAR_INPUT
      "PwrSuppOK" { ExternalAccessible := 'True'; ExternalVisible := 'False'; ExternalWritable := 'False'; } : BOOL;   //EPICS Status variable: PwrSuppOK
      "EnCmdR" { ExternalAccessible := 'True'; ExternalVisible := 'False'; ExternalWritable := 'False'; } : BOOL;   //EPICS Status variable: EnCmdR
   EPICSToPLCLength { ExternalAccessible := 'False'; ExternalVisible := 'False'; ExternalWritable := 'False'; } : Int;   // Length of device command register array (in words)
   EPICSToPLCDataBlockOffset { ExternalAccessible := 'False'; ExternalVisible := 'False'; ExternalWritable := 'False'; } : Int;   // Offset in EPICS->PLC comms block where this device data resides (in words)
   EPICSToPLCParametersStart { ExternalAccessible := 'False'; ExternalVisible := 'False'; ExternalWritable := 'False'; } : Int;   // The border offset between the Command and the Parameter area
   PLCToEPICSLength { ExternalAccessible := 'False'; ExternalVisible := 'False'; ExternalWritable := 'False'; } : Int;   // Length of device status register array (in words)
   PLCToEPICSDataBlockOffset { ExternalAccessible := 'False'; ExternalVisible := 'False'; ExternalWritable := 'False'; } : Int;   // Offset in PLC->EPICS comms block where this device data resides (in words)
   END_VAR
   VAR_OUTPUT
      DEVICE_PARAM_OK { ExternalAccessible := 'False'; ExternalVisible := 'False'; ExternalWritable := 'False'; } : Bool;
   END_VAR
   VAR_IN_OUT
   END_VAR
   Var DB_SPECIFIC
      MyWord { ExternalAccessible := 'False'; ExternalVisible := 'False'; ExternalWritable := 'False'; } : Word;
      MyBytesinWord { ExternalAccessible := 'False'; ExternalVisible := 'False'; ExternalWritable := 'False'; } AT MyWord : Array[0..1] of Byte;
      MyBoolsinWord { ExternalAccessible := 'False'; ExternalVisible := 'False'; ExternalWritable := 'False'; } AT MyWord : Array[0..15] of Bool;
      MyDInt { ExternalAccessible := 'False'; ExternalVisible := 'False'; ExternalWritable := 'False'; } : DInt;
      MyWordsinDint { ExternalAccessible := 'False'; ExternalVisible := 'False'; ExternalWritable := 'False'; } AT MyDInt : Array[0..1] of Word;
      MyReal { ExternalAccessible := 'False'; ExternalVisible := 'False'; ExternalWritable := 'False'; } : Real;
      MyWordsinReal { ExternalAccessible := 'False'; ExternalVisible := 'False'; ExternalWritable := 'False'; } AT MyReal : Array[0..1] of Word;
      MyInt { ExternalAccessible := 'False'; ExternalVisible := 'False'; ExternalWritable := 'False'; } : Int;
      MyWordinInt { ExternalAccessible := 'False'; ExternalVisible := 'False'; ExternalWritable := 'False'; } AT MyInt : Word;
      MyDWord { ExternalAccessible := 'False'; ExternalVisible := 'False'; ExternalWritable := 'False'; } : DWord;
      MyWordsinDWord { ExternalAccessible := 'False'; ExternalVisible := 'False'; ExternalWritable := 'False'; } AT MyDWord : Array[0..1] of Word;
      MyTime { ExternalAccessible := 'False'; ExternalVisible := 'False'; ExternalWritable := 'False'; } : Time;
      MyWordsinTime { ExternalAccessible := 'False'; ExternalVisible := 'False'; ExternalWritable := 'False'; } AT MyTime : Array[0..1] of Word;
      MyString { ExternalAccessible := 'False'; ExternalVisible := 'False'; ExternalWritable := 'False'; } : String[40];
      MyWordsinString { ExternalAccessible := 'False'; ExternalVisible := 'False'; ExternalWritable := 'False'; } AT MyString : Array[0..20] of Word;
   END_VAR
   VAR_TEMP
      HashModbus : DInt;
      HashIFA : DInt;
      HashTIAMap : DInt;
      i : Int;
   END_VAR
    //Author: Miklos Boros (miklos.boros@esss.se), Copyrigth 2017-2019 by European Spallation Source, Lund
    //This block was generated by PLCFactory, please don't change it MANUALLY!
    //Input File Name: ISrc-010_Ctrl-PLC-01-template-IFA-20191106135317.ifa
    //Generated: 20191106135317
    //According to HASH: 1347332123
    //Device type: ISRC_LEBT_PS_COIL
    //Description: This function does the variable mapping for a device. All device-variable will be linked to an interface variable defined in this block.

    //********************************************
    //****************HASH check******************
    //********************************************


    #MyWordsinDint[0] := "EPICSToPLC"."Word"[0];
    #MyWordsinDint[1] := "EPICSToPLC"."Word"[1];
    #HashModbus := #MyDInt; //Hash from EPICS/ModbusTCP

    #HashIFA := 1347332123; //Hash from Interface Factory as a constant

    #MyWordsinDint[0] := "PLCToEPICS"."Word"[0];
    #MyWordsinDint[1] := "PLCToEPICS"."Word"[1];
    #HashTIAMap := #MyDInt; //Hash from PLCFactory TIA Map


    IF ((#HashIFA = #HashModbus) AND (#HashModbus = #HashTIAMap)) THEN //Check CRCs
        #DEVICE_PARAM_OK := TRUE;
       //###########################  ISRC_LEBT Coil Power Supply  ##############################
       //###########################
       //STATUS BLOCK
       //###########################

    //********************************************
    //*************STATUS VARIABLES***************
    //********************************************


       #MyWord := W#0;
       #MyBoolsinWord[8] := #"PwrSuppOK";    //EPICSName: PwrSuppOK
       #MyBoolsinWord[9] := #"EnCmdR";    //EPICSName: EnCmdR
       "PLCToEPICS"."Word"[#PLCToEPICSDataBlockOffset + 0] := #MyWord;
    Else
       #DEVICE_PARAM_OK := FALSE; //Invalid Hash
    END_IF;
END_FUNCTION_BLOCK
FUNCTION_BLOCK "DEVTYPE_ISRC_LEBT_PS_REP"
{ S7_Optimized_Access := 'TRUE' }
VERSION : 1.0
   VAR_INPUT
      "VolOK" { ExternalAccessible := 'True'; ExternalVisible := 'False'; ExternalWritable := 'False'; } : BOOL;   //EPICS Status variable: VolOK
   EPICSToPLCLength { ExternalAccessible := 'False'; ExternalVisible := 'False'; ExternalWritable := 'False'; } : Int;   // Length of device command register array (in words)
   EPICSToPLCDataBlockOffset { ExternalAccessible := 'False'; ExternalVisible := 'False'; ExternalWritable := 'False'; } : Int;   // Offset in EPICS->PLC comms block where this device data resides (in words)
   EPICSToPLCParametersStart { ExternalAccessible := 'False'; ExternalVisible := 'False'; ExternalWritable := 'False'; } : Int;   // The border offset between the Command and the Parameter area
   PLCToEPICSLength { ExternalAccessible := 'False'; ExternalVisible := 'False'; ExternalWritable := 'False'; } : Int;   // Length of device status register array (in words)
   PLCToEPICSDataBlockOffset { ExternalAccessible := 'False'; ExternalVisible := 'False'; ExternalWritable := 'False'; } : Int;   // Offset in PLC->EPICS comms block where this device data resides (in words)
   END_VAR
   VAR_OUTPUT
      "iVolR" { ExternalAccessible := 'True'; ExternalVisible := 'False'; ExternalWritable := 'False'; } : REAL;   //EPICS Parameter variable: iVolR
      DEVICE_PARAM_OK { ExternalAccessible := 'False'; ExternalVisible := 'False'; ExternalWritable := 'False'; } : Bool;
   END_VAR
   VAR_IN_OUT
   END_VAR
   Var DB_SPECIFIC
      MyWord { ExternalAccessible := 'False'; ExternalVisible := 'False'; ExternalWritable := 'False'; } : Word;
      MyBytesinWord { ExternalAccessible := 'False'; ExternalVisible := 'False'; ExternalWritable := 'False'; } AT MyWord : Array[0..1] of Byte;
      MyBoolsinWord { ExternalAccessible := 'False'; ExternalVisible := 'False'; ExternalWritable := 'False'; } AT MyWord : Array[0..15] of Bool;
      MyDInt { ExternalAccessible := 'False'; ExternalVisible := 'False'; ExternalWritable := 'False'; } : DInt;
      MyWordsinDint { ExternalAccessible := 'False'; ExternalVisible := 'False'; ExternalWritable := 'False'; } AT MyDInt : Array[0..1] of Word;
      MyReal { ExternalAccessible := 'False'; ExternalVisible := 'False'; ExternalWritable := 'False'; } : Real;
      MyWordsinReal { ExternalAccessible := 'False'; ExternalVisible := 'False'; ExternalWritable := 'False'; } AT MyReal : Array[0..1] of Word;
      MyInt { ExternalAccessible := 'False'; ExternalVisible := 'False'; ExternalWritable := 'False'; } : Int;
      MyWordinInt { ExternalAccessible := 'False'; ExternalVisible := 'False'; ExternalWritable := 'False'; } AT MyInt : Word;
      MyDWord { ExternalAccessible := 'False'; ExternalVisible := 'False'; ExternalWritable := 'False'; } : DWord;
      MyWordsinDWord { ExternalAccessible := 'False'; ExternalVisible := 'False'; ExternalWritable := 'False'; } AT MyDWord : Array[0..1] of Word;
      MyTime { ExternalAccessible := 'False'; ExternalVisible := 'False'; ExternalWritable := 'False'; } : Time;
      MyWordsinTime { ExternalAccessible := 'False'; ExternalVisible := 'False'; ExternalWritable := 'False'; } AT MyTime : Array[0..1] of Word;
      MyString { ExternalAccessible := 'False'; ExternalVisible := 'False'; ExternalWritable := 'False'; } : String[40];
      MyWordsinString { ExternalAccessible := 'False'; ExternalVisible := 'False'; ExternalWritable := 'False'; } AT MyString : Array[0..20] of Word;
   END_VAR
   VAR_TEMP
      HashModbus : DInt;
      HashIFA : DInt;
      HashTIAMap : DInt;
      i : Int;
   END_VAR
    //Author: Miklos Boros (miklos.boros@esss.se), Copyrigth 2017-2019 by European Spallation Source, Lund
    //This block was generated by PLCFactory, please don't change it MANUALLY!
    //Input File Name: ISrc-010_Ctrl-PLC-01-template-IFA-20191106135317.ifa
    //Generated: 20191106135317
    //According to HASH: 1347332123
    //Device type: ISRC_LEBT_PS_REP
    //Description: This function does the variable mapping for a device. All device-variable will be linked to an interface variable defined in this block.

    //********************************************
    //****************HASH check******************
    //********************************************


    #MyWordsinDint[0] := "EPICSToPLC"."Word"[0];
    #MyWordsinDint[1] := "EPICSToPLC"."Word"[1];
    #HashModbus := #MyDInt; //Hash from EPICS/ModbusTCP

    #HashIFA := 1347332123; //Hash from Interface Factory as a constant

    #MyWordsinDint[0] := "PLCToEPICS"."Word"[0];
    #MyWordsinDint[1] := "PLCToEPICS"."Word"[1];
    #HashTIAMap := #MyDInt; //Hash from PLCFactory TIA Map


    IF ((#HashIFA = #HashModbus) AND (#HashModbus = #HashTIAMap)) THEN //Check CRCs
        #DEVICE_PARAM_OK := TRUE;
       //###########################  ISrc and LEBT Repeller's Power Supply  ##############################
       //###########################
       //STATUS BLOCK
       //###########################

    //********************************************
    //*************STATUS VARIABLES***************
    //********************************************


       #MyWord := W#0;
       #MyBoolsinWord[8] := #"VolOK";    //EPICSName: VolOK
       "PLCToEPICS"."Word"[#PLCToEPICSDataBlockOffset + 0] := #MyWord;

    //********************************************
    //************PARAMETER VARIABLES*************
    //********************************************


